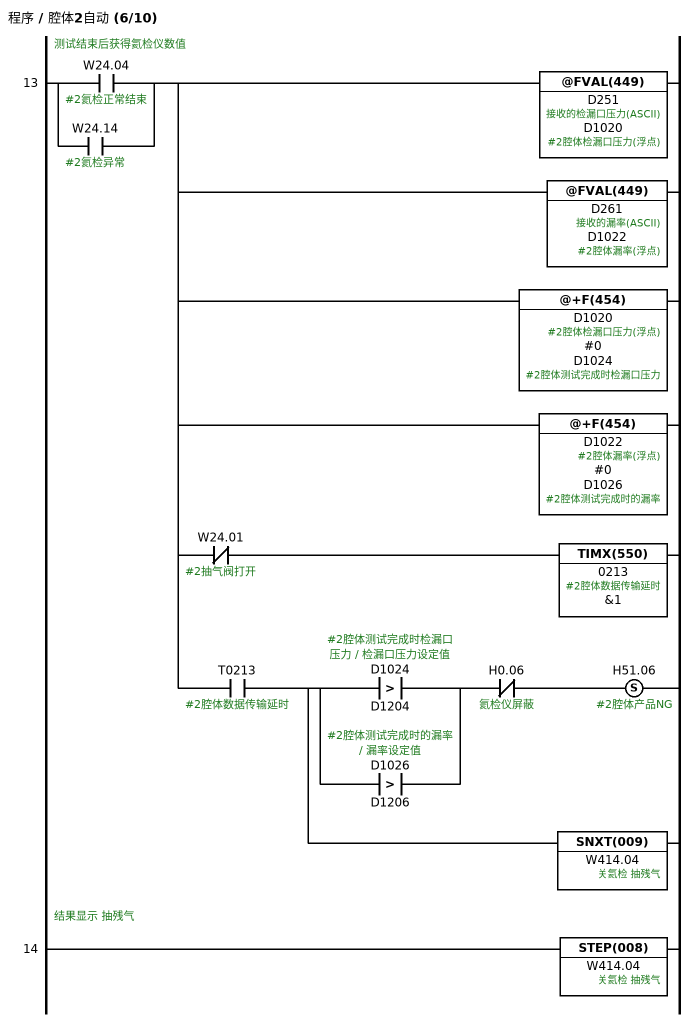
; [picture p72: 程序 / 腔体2自动, rungs 13-14]
; rung 13: 测试结束后获得氦检仪数值
LD W24.04  ; #2氦检正常结束
OR W24.14  ; #2氦检异常
OUT TR0
@FVAL(449) D251 D1020  ; 接收的检漏口压力(ASCII), #2腔体检漏口压力(浮点)
@FVAL(449) D261 D1022  ; 接收的漏率(ASCII), #2腔体漏率(浮点)
@+F(454) D1020 #0 D1024  ; #2腔体检漏口压力(浮点), #2腔体测试完成时检漏口压力
@+F(454) D1022 #0 D1026  ; #2腔体漏率(浮点), #2腔体测试完成时的漏率
ANDNOT W24.01  ; #2抽气阀打开
TIMX(550) 0213 &1  ; #2腔体数据传输延时
LD TR0
AND T0213  ; #2腔体数据传输延时
OUT TR0
LD>F(333) D1024 D1204  ; #2腔体测试完成时检漏口压力, 检漏口压力设定值
OR>F(333) D1026 D1206  ; #2腔体测试完成时的漏率, 漏率设定值
ANDLD
ANDNOT H0.06  ; 氦检仪屏蔽
SET H51.06  ; #2腔体产品NG
LD TR0
SNXT(009) W414.04  ; 关氦检 抽残气
; rung 14: 结果显示 抽残气
STEP(008) W414.04  ; 关氦检 抽残气

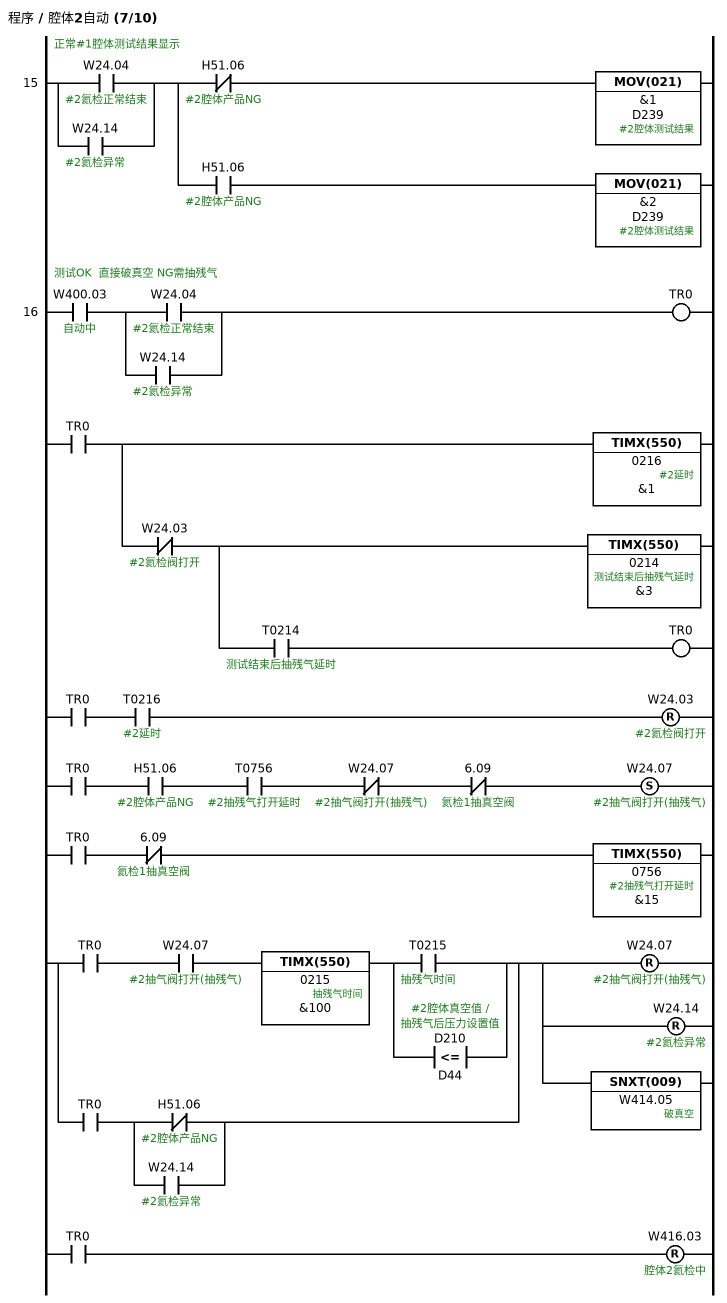
; rung 15: 正常#1腔体测试结果显示
LD W24.04  ; #2氦检正常结束
OR W24.14  ; #2氦检异常
OUT TR0
ANDNOT H51.06  ; #2腔体产品NG
MOV(021) &1 D239  ; #2腔体测试结果
LD TR0
AND H51.06  ; #2腔体产品NG
MOV(021) &2 D239  ; #2腔体测试结果
; rung 16: 测试OK  直接破真空 NG需抽残气
LD W400.03  ; 自动中
LD W24.04  ; #2氦检正常结束
OR W24.14  ; #2氦检异常
ANDLD
OUT TR0
AND T0216  ; #2延时
RSET W24.03  ; #2氦检阀打开
LD TR0
TIMX(550) 0216 &1  ; #2延时
ANDNOT W24.03  ; #2氦检阀打开
TIMX(550) 0214 &3  ; 测试结束后抽残气延时
AND T0214  ; 测试结束后抽残气延时
OUT TR0
AND H51.06  ; #2腔体产品NG
AND T0756  ; #2抽残气打开延时
ANDNOT W24.07  ; #2抽气阀打开(抽残气)
ANDNOT 6.09  ; 氦检1抽真空阀
SET W24.07  ; #2抽气阀打开(抽残气)
LD TR0
ANDNOT 6.09  ; 氦检1抽真空阀
TIMX(550) 0756 &15  ; #2抽残气打开延时
LD TR0
AND W24.07  ; #2抽气阀打开(抽残气)
TIMX(550) 0215 &100  ; 抽残气时间
LD T0215  ; 抽残气时间
OR<=F(332) D210 D44  ; #2腔体真空值, 抽残气后压力设置值
ANDLD
LD TR0
LDNOT H51.06  ; #2腔体产品NG
OR W24.14  ; #2氦检异常
ANDLD
ORLD
RSET W24.07  ; #2抽气阀打开(抽残气)
RSET W24.14  ; #2氦检异常
SNXT(009) W414.05  ; 破真空
LD TR0
RSET W416.03  ; 腔体2氦检中

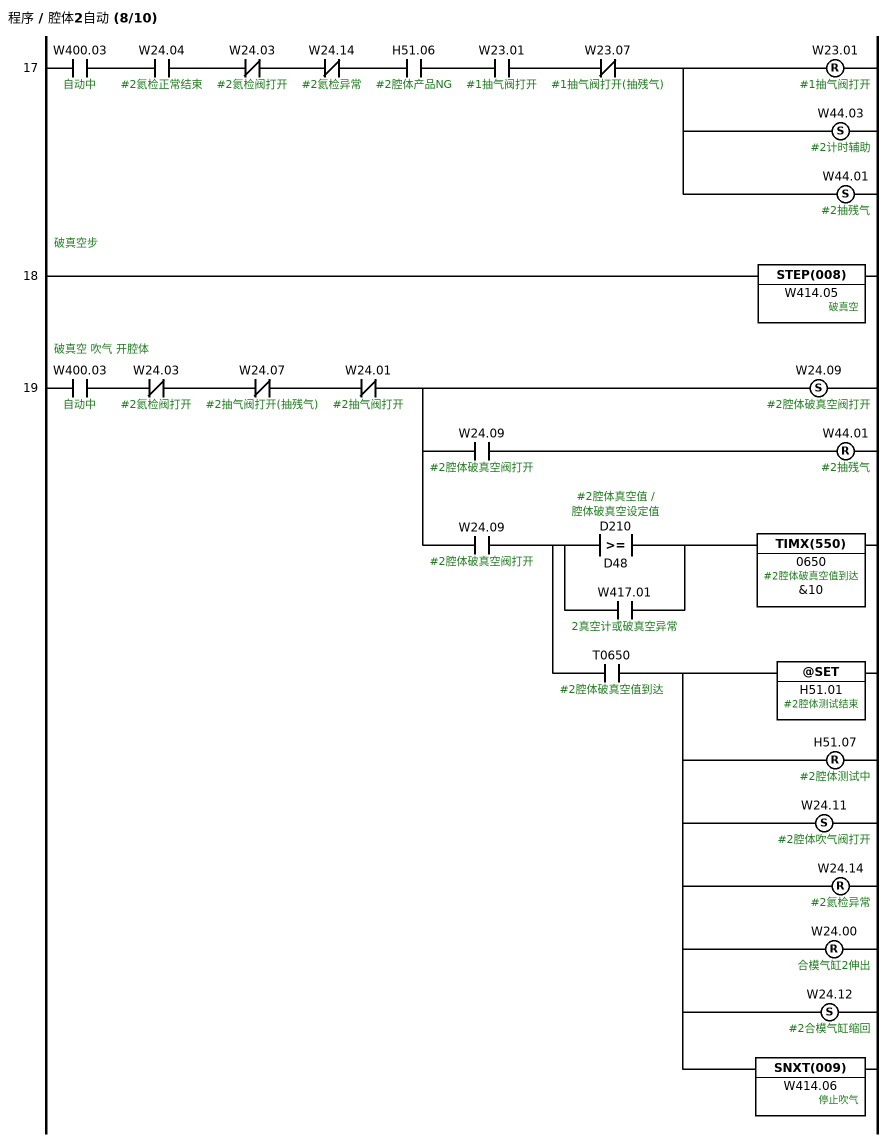
; rung 17
LD W400.03  ; 自动中
AND W24.04  ; #2氦检正常结束
ANDNOT W24.03  ; #2氦检阀打开
ANDNOT W24.14  ; #2氦检异常
AND H51.06  ; #2腔体产品NG
AND W23.01  ; #1抽气阀打开
ANDNOT W23.07  ; #1抽气阀打开(抽残气)
RSET W23.01  ; #1抽气阀打开
SET W44.03  ; #2计时辅助
SET W44.01  ; #2抽残气
; rung 18: 破真空步
STEP(008) W414.05  ; 破真空
; rung 19: 破真空 吹气 开腔体
LD W400.03  ; 自动中
ANDNOT W24.03  ; #2氦检阀打开
ANDNOT W24.07  ; #2抽气阀打开(抽残气)
ANDNOT W24.01  ; #2抽气阀打开
OUT TR0
SET W24.09  ; #2腔体破真空阀打开
AND W24.09  ; #2腔体破真空阀打开
RSET W44.01  ; #2抽残气
LD TR0
AND W24.09  ; #2腔体破真空阀打开
OUT TR0
LD>=F(334) D210 D48  ; #2腔体真空值, 腔体破真空设定值
OR W417.01  ; 2真空计或破真空异常
ANDLD
TIMX(550) 0650 &10  ; #2腔体破真空值到达
LD TR0
AND T0650  ; #2腔体破真空值到达
@SET H51.01  ; #2腔体测试结束
RSET H51.07  ; #2腔体测试中
SET W24.11  ; #2腔体吹气阀打开
RSET W24.14  ; #2氦检异常
RSET W24.00  ; 合模气缸2伸出
SET W24.12  ; #2合模气缸缩回
SNXT(009) W414.06  ; 停止吹气

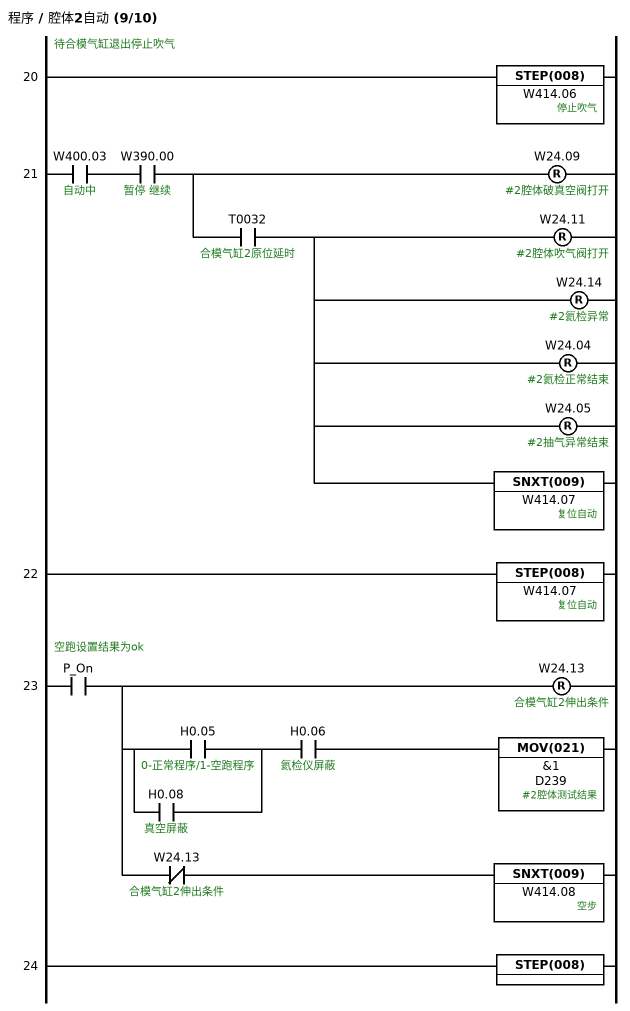
; rung 20: 待合模气缸退出停止吹气
STEP(008) W414.06  ; 停止吹气
; rung 21
LD W400.03  ; 自动中
AND W390.00  ; 暂停 继续
RSET W24.09  ; #2腔体破真空阀打开
AND T0032  ; 合模气缸2原位延时
RSET W24.11  ; #2腔体吹气阀打开
RSET W24.14  ; #2氦检异常
RSET W24.04  ; #2氦检正常结束
RSET W24.05  ; #2抽气异常结束
SNXT(009) W414.07  ; 复位自动
; rung 22
STEP(008) W414.07  ; 复位自动
; rung 23: 空跑设置结果为ok
LD P_On
OUT TR0
RSET W24.13  ; 合模气缸2伸出条件
LD H0.05  ; 0-正常程序/1-空跑程序
OR H0.08  ; 真空屏蔽
ANDLD
AND H0.06  ; 氦检仪屏蔽
MOV(021) &1 D239  ; #2腔体测试结果
LD TR0
ANDNOT W24.13  ; 合模气缸2伸出条件
SNXT(009) W414.08  ; 空步
; rung 24
STEP(008)

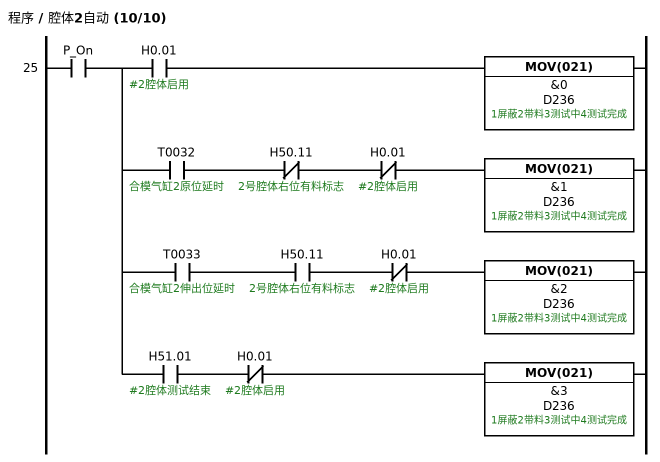
; rung 25
LD P_On
OUT TR0
AND H0.01  ; #2腔体启用
MOV(021) &0 D236  ; 1屏蔽2带料3测试中4测试完成
LD TR0
AND T0032  ; 合模气缸2原位延时
ANDNOT H50.11  ; 2号腔体右位有料标志
ANDNOT H0.01  ; #2腔体启用
MOV(021) &1 D236  ; 1屏蔽2带料3测试中4测试完成
LD TR0
AND T0033  ; 合模气缸2伸出位延时
AND H50.11  ; 2号腔体右位有料标志
ANDNOT H0.01  ; #2腔体启用
MOV(021) &2 D236  ; 1屏蔽2带料3测试中4测试完成
LD TR0
AND H51.01  ; #2腔体测试结束
ANDNOT H0.01  ; #2腔体启用
MOV(021) &3 D236  ; 1屏蔽2带料3测试中4测试完成

### Section 下料轴自动

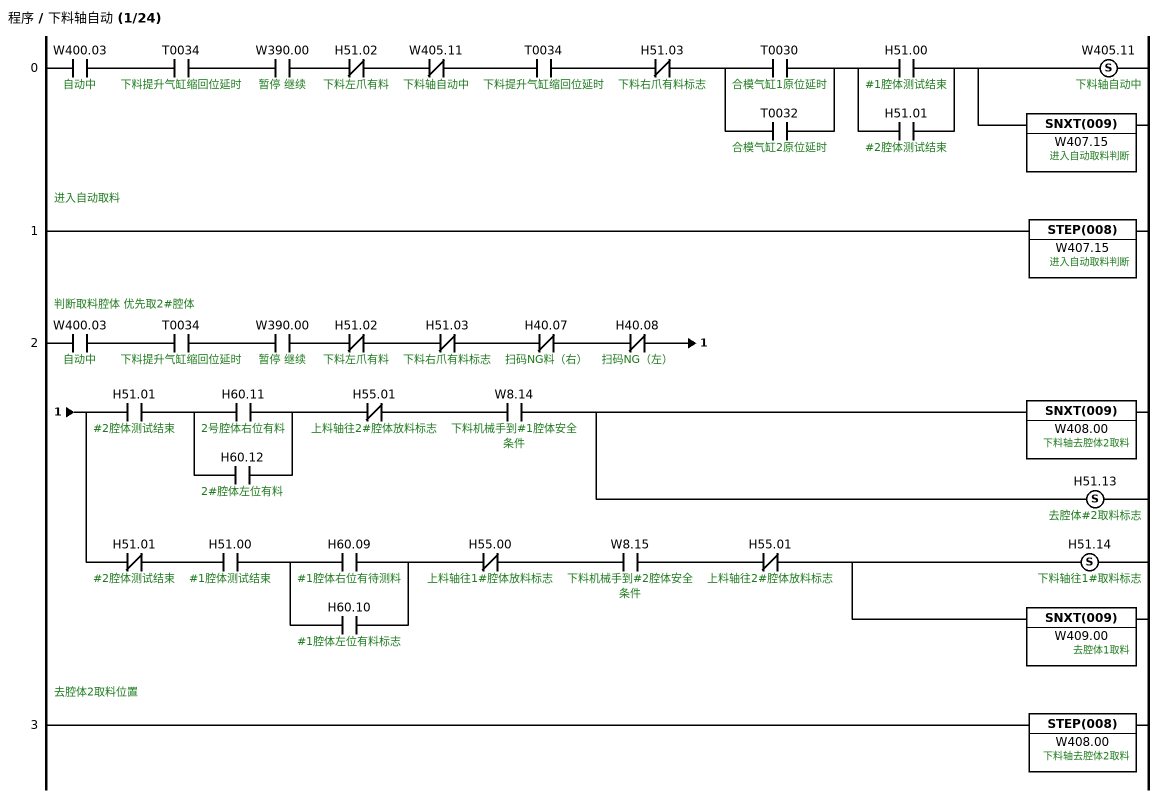
; rung 0
LD W400.03  ; 自动中
AND T0034  ; 下料提升气缸缩回位延时
AND W390.00  ; 暂停 继续
ANDNOT H51.02  ; 下料左爪有料
ANDNOT W405.11  ; 下料轴自动中
AND T0034  ; 下料提升气缸缩回位延时
ANDNOT H51.03  ; 下料右爪有料标志
LD T0030  ; 合模气缸1原位延时
OR T0032  ; 合模气缸2原位延时
ANDLD
LD H51.00  ; #1腔体测试结束
OR H51.01  ; #2腔体测试结束
ANDLD
SET W405.11  ; 下料轴自动中
SNXT(009) W407.15  ; 进入自动取料判断
; rung 1: 进入自动取料
STEP(008) W407.15  ; 进入自动取料判断
; rung 2: 判断取料腔体 优先取2#腔体
LD W400.03  ; 自动中
AND T0034  ; 下料提升气缸缩回位延时
AND W390.00  ; 暂停 继续
ANDNOT H51.02  ; 下料左爪有料
ANDNOT H51.03  ; 下料右爪有料标志
ANDNOT H40.07  ; 扫码NG料（右）
ANDNOT H40.08  ; 扫码NG（左）
OUT TR0
AND H51.01  ; #2腔体测试结束
LD H60.11  ; 2号腔体右位有料
OR H60.12  ; 2#腔体左位有料
ANDLD
ANDNOT H55.01  ; 上料轴往2#腔体放料标志
AND W8.14  ; 下料机械手到#1腔体安全条件
SNXT(009) W408.00  ; 下料轴去腔体2取料
SET H51.13  ; 去腔体#2取料标志
LD TR0
ANDNOT H51.01  ; #2腔体测试结束
AND H51.00  ; #1腔体测试结束
LD H60.09  ; #1腔体右位有待测料
OR H60.10  ; #1腔体左位有料标志
ANDLD
ANDNOT H55.00  ; 上料轴往1#腔体放料标志
AND W8.15  ; 下料机械手到#2腔体安全条件
ANDNOT H55.01  ; 上料轴往2#腔体放料标志
SET H51.14  ; 下料轴往1#取料标志
SNXT(009) W409.00  ; 去腔体1取料
; rung 3: 去腔体2取料位置
STEP(008) W408.00  ; 下料轴去腔体2取料

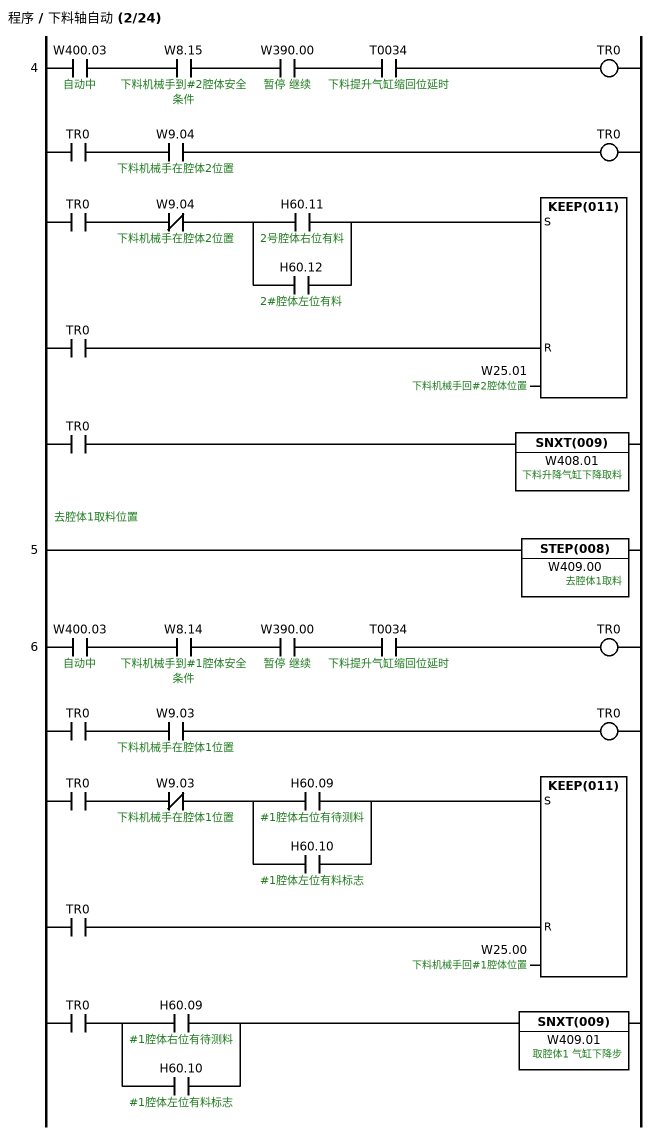
; rung 4
LD W400.03  ; 自动中
AND W8.15  ; 下料机械手到#2腔体安全条件
AND W390.00  ; 暂停 继续
AND T0034  ; 下料提升气缸缩回位延时
OUT TR0
ANDNOT W9.04  ; 下料机械手在腔体2位置
LD H60.11  ; 2号腔体右位有料
OR H60.12  ; 2#腔体左位有料
ANDLD
LD TR0
AND W9.04  ; 下料机械手在腔体2位置
OUT TR0
KEEP(011) W25.01  ; 下料机械手回#2腔体位置
LD TR0
SNXT(009) W408.01  ; 下料升降气缸下降取料
; rung 5: 去腔体1取料位置
STEP(008) W409.00  ; 去腔体1取料
; rung 6
LD W400.03  ; 自动中
AND W8.14  ; 下料机械手到#1腔体安全条件
AND W390.00  ; 暂停 继续
AND T0034  ; 下料提升气缸缩回位延时
OUT TR0
ANDNOT W9.03  ; 下料机械手在腔体1位置
LD H60.09  ; #1腔体右位有待测料
OR H60.10  ; #1腔体左位有料标志
ANDLD
LD TR0
AND W9.03  ; 下料机械手在腔体1位置
OUT TR0
KEEP(011) W25.00  ; 下料机械手回#1腔体位置
LD TR0
LD H60.09  ; #1腔体右位有待测料
OR H60.10  ; #1腔体左位有料标志
ANDLD
SNXT(009) W409.01  ; 取腔体1 气缸下降步

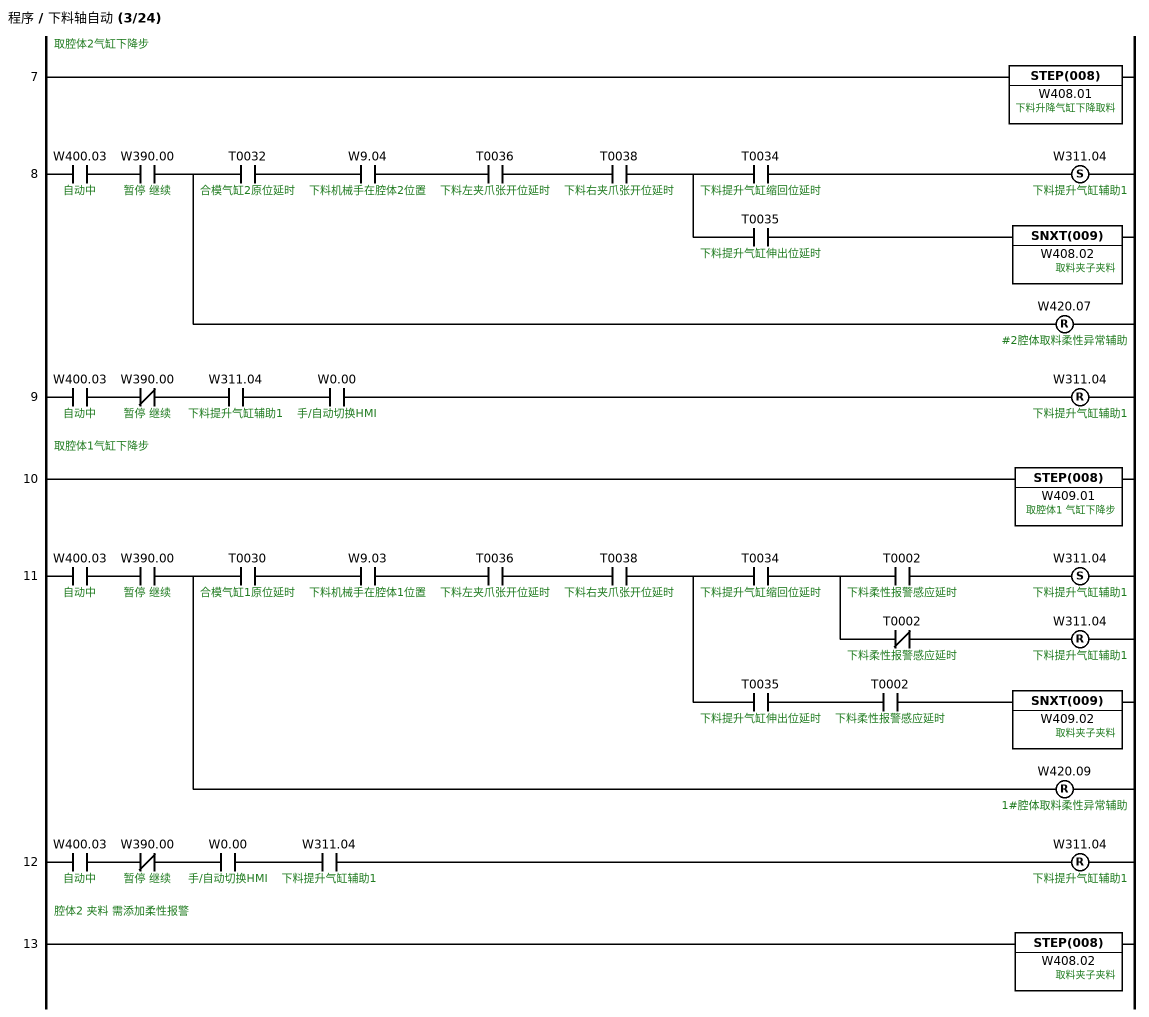
; rung 7: 取腔体2气缸下降步
STEP(008) W408.01  ; 下料升降气缸下降取料
; rung 8
LD W400.03  ; 自动中
AND W390.00  ; 暂停 继续
OUT TR0
AND T0032  ; 合模气缸2原位延时
AND W9.04  ; 下料机械手在腔体2位置
AND T0036  ; 下料左夹爪张开位延时
AND T0038  ; 下料右夹爪张开位延时
OUT TR1
AND T0034  ; 下料提升气缸缩回位延时
SET W311.04  ; 下料提升气缸辅助1
LD TR1
AND T0035  ; 下料提升气缸伸出位延时
SNXT(009) W408.02  ; 取料夹子夹料
LD TR0
RSET W420.07  ; #2腔体取料柔性异常辅助
; rung 9
LD W400.03  ; 自动中
ANDNOT W390.00  ; 暂停 继续
AND W311.04  ; 下料提升气缸辅助1
AND W0.00  ; 手/自动切换HMI
RSET W311.04  ; 下料提升气缸辅助1
; rung 10: 取腔体1气缸下降步
STEP(008) W409.01  ; 取腔体1 气缸下降步
; rung 11
LD W400.03  ; 自动中
AND W390.00  ; 暂停 继续
OUT TR0
AND T0030  ; 合模气缸1原位延时
AND W9.03  ; 下料机械手在腔体1位置
AND T0036  ; 下料左夹爪张开位延时
AND T0038  ; 下料右夹爪张开位延时
OUT TR1
AND T0034  ; 下料提升气缸缩回位延时
OUT TR2
AND T0002  ; 下料柔性报警感应延时
SET W311.04  ; 下料提升气缸辅助1
LD TR2
ANDNOT T0002  ; 下料柔性报警感应延时
RSET W311.04  ; 下料提升气缸辅助1
LD TR1
AND T0035  ; 下料提升气缸伸出位延时
AND T0002  ; 下料柔性报警感应延时
SNXT(009) W409.02  ; 取料夹子夹料
LD TR0
RSET W420.09  ; 1#腔体取料柔性异常辅助
; rung 12
LD W400.03  ; 自动中
ANDNOT W390.00  ; 暂停 继续
AND W0.00  ; 手/自动切换HMI
AND W311.04  ; 下料提升气缸辅助1
RSET W311.04  ; 下料提升气缸辅助1
; rung 13: 腔体2 夹料 需添加柔性报警
STEP(008) W408.02  ; 取料夹子夹料

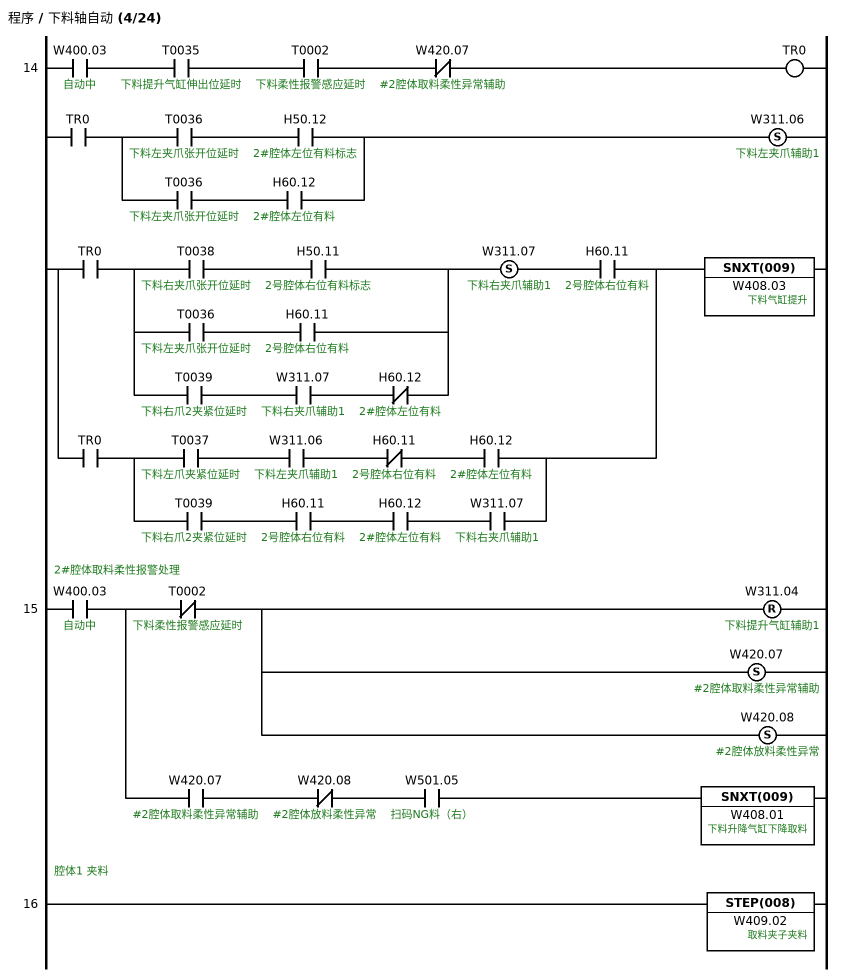
; rung 14
LD W400.03  ; 自动中
AND T0035  ; 下料提升气缸伸出位延时
AND T0002  ; 下料柔性报警感应延时
ANDNOT W420.07  ; #2腔体取料柔性异常辅助
OUT TR0
LD T0036  ; 下料左夹爪张开位延时
AND H50.12  ; 2#腔体左位有料标志
LD T0036  ; 下料左夹爪张开位延时
AND H60.12  ; 2#腔体左位有料
ORLD
ANDLD
SET W311.06  ; 下料左夹爪辅助1
LD TR0
LD T0038  ; 下料右夹爪张开位延时
AND H50.11  ; 2号腔体右位有料标志
LD T0036  ; 下料左夹爪张开位延时
AND H60.11  ; 2号腔体右位有料
ORLD
LD T0039  ; 下料右爪2夹紧位延时
AND W311.07  ; 下料右夹爪辅助1
ANDNOT H60.12  ; 2#腔体左位有料
ORLD
ANDLD
SET W311.07  ; 下料右夹爪辅助1
AND H60.11  ; 2号腔体右位有料
LD TR0
LD T0037  ; 下料左爪夹紧位延时
AND W311.06  ; 下料左夹爪辅助1
ANDNOT H60.11  ; 2号腔体右位有料
AND H60.12  ; 2#腔体左位有料
LD T0039  ; 下料右爪2夹紧位延时
AND H60.11  ; 2号腔体右位有料
AND H60.12  ; 2#腔体左位有料
AND W311.07  ; 下料右夹爪辅助1
ORLD
ANDLD
ORLD
SNXT(009) W408.03  ; 下料气缸提升
; rung 15: 2#腔体取料柔性报警处理
LD W400.03  ; 自动中
OUT TR0
ANDNOT T0002  ; 下料柔性报警感应延时
RSET W311.04  ; 下料提升气缸辅助1
SET W420.07  ; #2腔体取料柔性异常辅助
SET W420.08  ; #2腔体放料柔性异常
LD TR0
AND W420.07  ; #2腔体取料柔性异常辅助
ANDNOT W420.08  ; #2腔体放料柔性异常
AND W501.05  ; 扫码NG料（右）
SNXT(009) W408.01  ; 下料升降气缸下降取料
; rung 16: 腔体1 夹料
STEP(008) W409.02  ; 取料夹子夹料

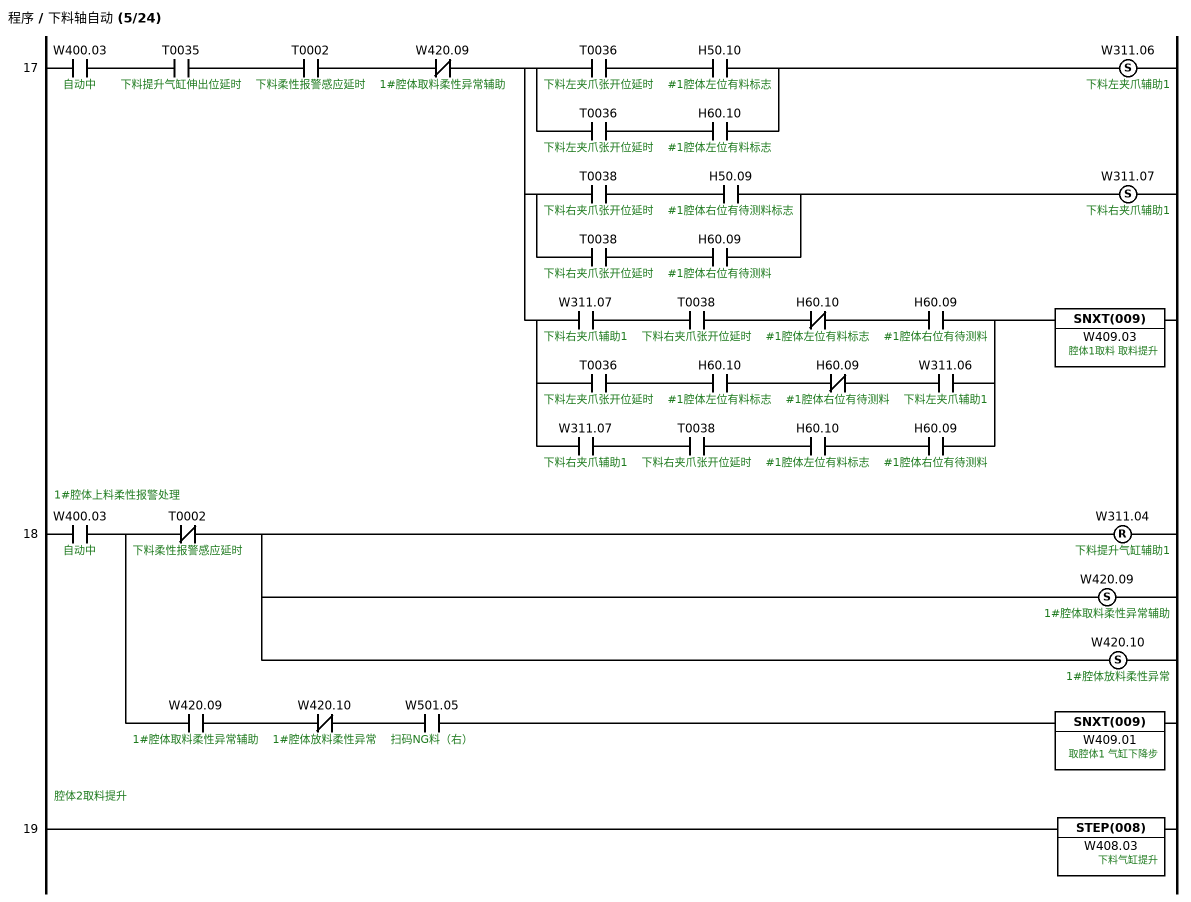
; rung 17
LD W400.03  ; 自动中
AND T0035  ; 下料提升气缸伸出位延时
AND T0002  ; 下料柔性报警感应延时
ANDNOT W420.09  ; 1#腔体取料柔性异常辅助
OUT TR0
LD T0036  ; 下料左夹爪张开位延时
AND H50.10  ; #1腔体左位有料标志
LD T0036  ; 下料左夹爪张开位延时
AND H60.10  ; #1腔体左位有料标志
ORLD
ANDLD
SET W311.06  ; 下料左夹爪辅助1
LD TR0
LD T0038  ; 下料右夹爪张开位延时
AND H50.09  ; #1腔体右位有待测料标志
LD T0038  ; 下料右夹爪张开位延时
AND H60.09  ; #1腔体右位有待测料
ORLD
ANDLD
SET W311.07  ; 下料右夹爪辅助1
LD TR0
LD W311.07  ; 下料右夹爪辅助1
AND T0038  ; 下料右夹爪张开位延时
ANDNOT H60.10  ; #1腔体左位有料标志
AND H60.09  ; #1腔体右位有待测料
LD T0036  ; 下料左夹爪张开位延时
AND H60.10  ; #1腔体左位有料标志
ANDNOT H60.09  ; #1腔体右位有待测料
AND W311.06  ; 下料左夹爪辅助1
ORLD
LD W311.07  ; 下料右夹爪辅助1
AND T0038  ; 下料右夹爪张开位延时
AND H60.10  ; #1腔体左位有料标志
AND H60.09  ; #1腔体右位有待测料
ORLD
ANDLD
SNXT(009) W409.03  ; 腔体1取料 取料提升
; rung 18: 1#腔体上料柔性报警处理
LD W400.03  ; 自动中
OUT TR0
ANDNOT T0002  ; 下料柔性报警感应延时
RSET W311.04  ; 下料提升气缸辅助1
SET W420.09  ; 1#腔体取料柔性异常辅助
SET W420.10  ; 1#腔体放料柔性异常
LD TR0
AND W420.09  ; 1#腔体取料柔性异常辅助
ANDNOT W420.10  ; 1#腔体放料柔性异常
AND W501.05  ; 扫码NG料（右）
SNXT(009) W409.01  ; 取腔体1 气缸下降步
; rung 19: 腔体2取料提升
STEP(008) W408.03  ; 下料气缸提升

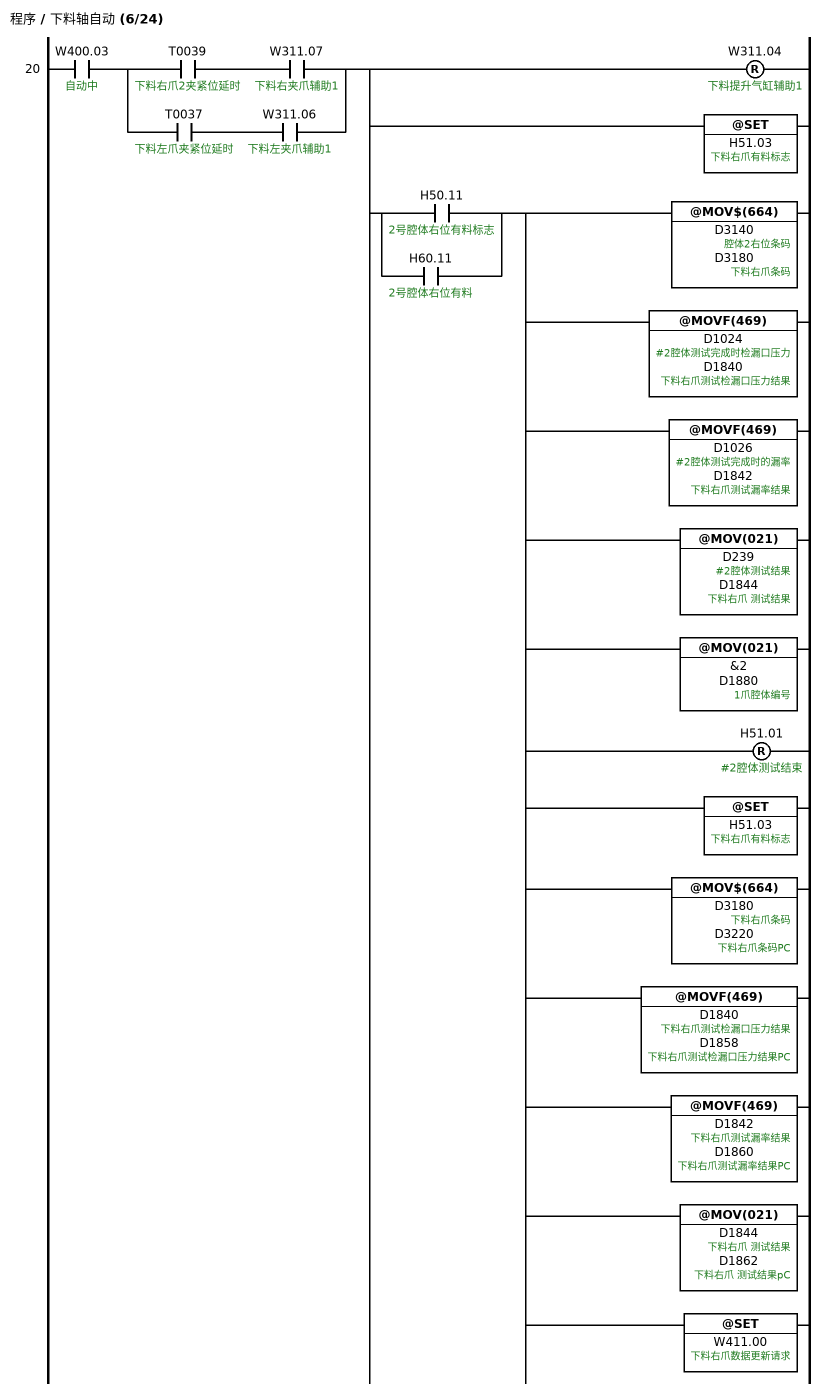

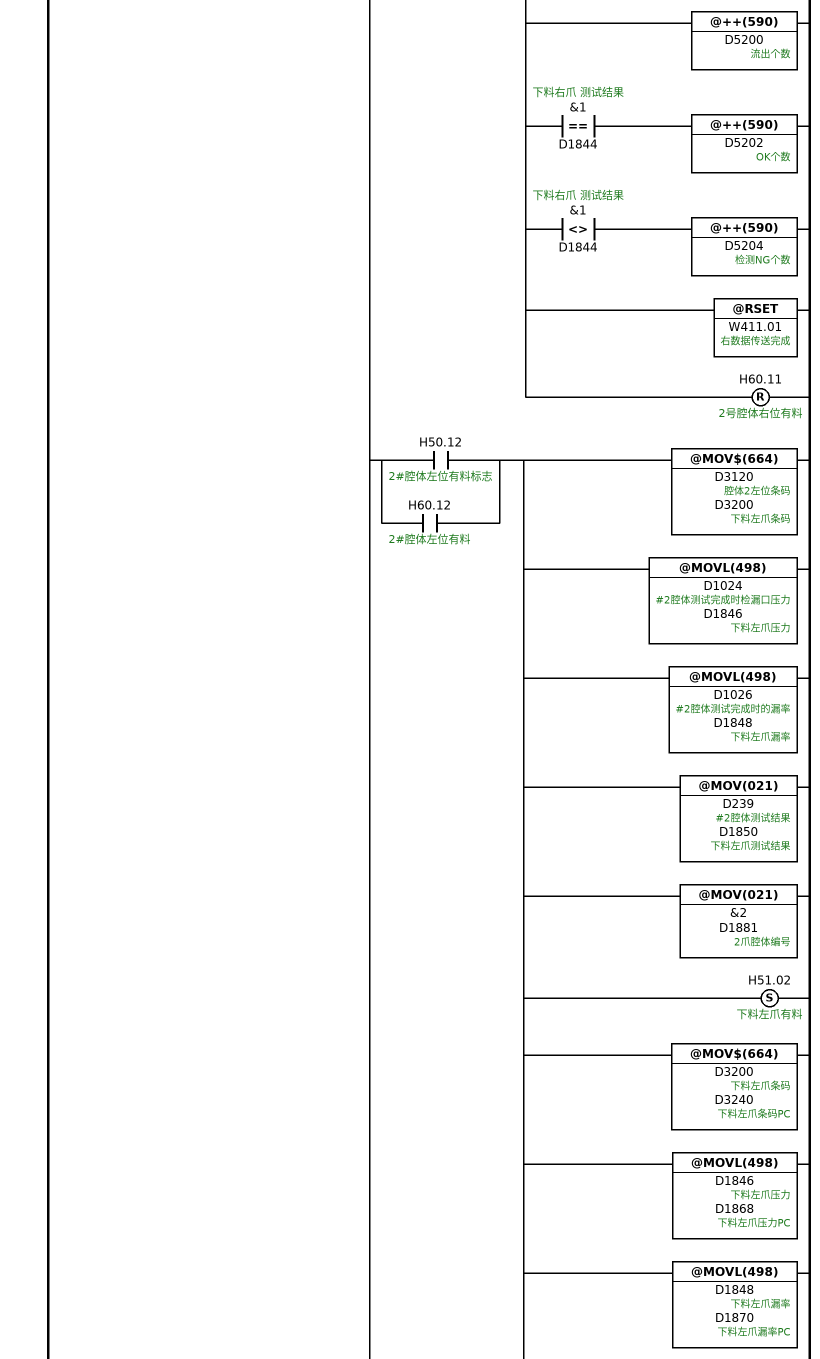

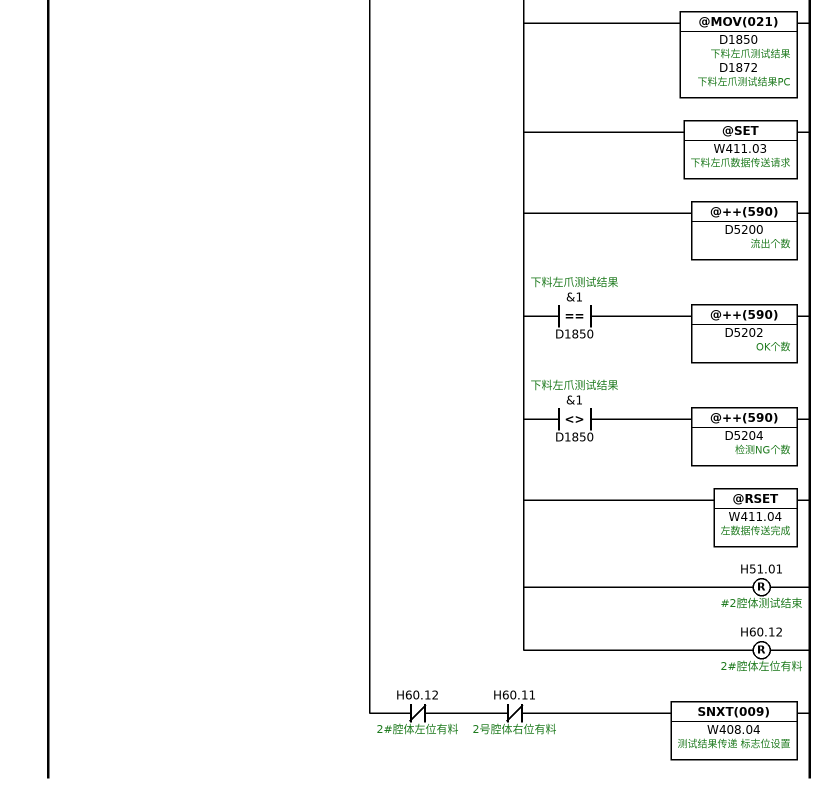
; rung 20
LD W400.03  ; 自动中
LD T0039  ; 下料右爪2夹紧位延时
AND W311.07  ; 下料右夹爪辅助1
LD T0037  ; 下料左爪夹紧位延时
AND W311.06  ; 下料左夹爪辅助1
ORLD
ANDLD
OUT TR0
RSET W311.04  ; 下料提升气缸辅助1
@SET H51.03  ; 下料右爪有料标志
LD H50.11  ; 2号腔体右位有料标志
OR H60.11  ; 2号腔体右位有料
ANDLD
OUT TR1
@MOV$(664) D3140 D3180  ; 腔体2右位条码, 下料右爪条码
@MOVF(469) D1024 D1840  ; #2腔体测试完成时检漏口压力, 下料右爪测试检漏口压力结果
@MOVF(469) D1026 D1842  ; #2腔体测试完成时的漏率, 下料右爪测试漏率结果
@MOV(021) D239 D1844  ; #2腔体测试结果, 下料右爪 测试结果
@MOV(021) &2 D1880  ; 1爪腔体编号
RSET H51.01  ; #2腔体测试结束
@SET H51.03  ; 下料右爪有料标志
@MOV$(664) D3180 D3220  ; 下料右爪条码, 下料右爪条码PC
@MOVF(469) D1840 D1858  ; 下料右爪测试检漏口压力结果, 下料右爪测试检漏口压力结果PC
@MOVF(469) D1842 D1860  ; 下料右爪测试漏率结果, 下料右爪测试漏率结果PC
@MOV(021) D1844 D1862  ; 下料右爪 测试结果, 下料右爪 测试结果pC
@SET W411.00  ; 下料右爪数据更新请求
@++(590) D5200  ; 流出个数
AND=(300) &1 D1844  ; 下料右爪 测试结果
@++(590) D5202  ; OK个数
LD TR1
AND<>(305) &1 D1844  ; 下料右爪 测试结果
@++(590) D5204  ; 检测NG个数
LD TR1
@RSET W411.01  ; 右数据传送完成
RSET H60.11  ; 2号腔体右位有料
LD TR0
LD H50.12  ; 2#腔体左位有料标志
OR H60.12  ; 2#腔体左位有料
ANDLD
OUT TR1
@MOV$(664) D3120 D3200  ; 腔体2左位条码, 下料左爪条码
@MOVL(498) D1024 D1846  ; #2腔体测试完成时检漏口压力, 下料左爪压力
@MOVL(498) D1026 D1848  ; #2腔体测试完成时的漏率, 下料左爪漏率
@MOV(021) D239 D1850  ; #2腔体测试结果, 下料左爪测试结果
@MOV(021) &2 D1881  ; 2爪腔体编号
SET H51.02  ; 下料左爪有料
@MOV$(664) D3200 D3240  ; 下料左爪条码, 下料左爪条码PC
@MOVL(498) D1846 D1868  ; 下料左爪压力, 下料左爪压力PC
@MOVL(498) D1848 D1870  ; 下料左爪漏率, 下料左爪漏率PC
@MOV(021) D1850 D1872  ; 下料左爪测试结果, 下料左爪测试结果PC
@SET W411.03  ; 下料左爪数据传送请求
@++(590) D5200  ; 流出个数
AND=(300) &1 D1850  ; 下料左爪测试结果
@++(590) D5202  ; OK个数
LD TR1
AND<>(305) &1 D1850  ; 下料左爪测试结果
@++(590) D5204  ; 检测NG个数
LD TR1
@RSET W411.04  ; 左数据传送完成
RSET H51.01  ; #2腔体测试结束
RSET H60.12  ; 2#腔体左位有料
LD TR0
ANDNOT H60.12  ; 2#腔体左位有料
ANDNOT H60.11  ; 2号腔体右位有料
SNXT(009) W408.04  ; 测试结果传递 标志位设置

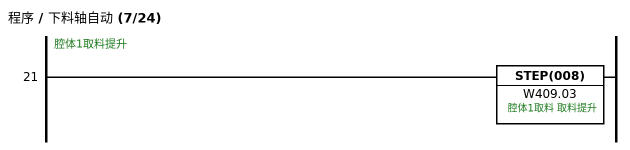
; rung 21: 腔体1取料提升
STEP(008) W409.03  ; 腔体1取料 取料提升

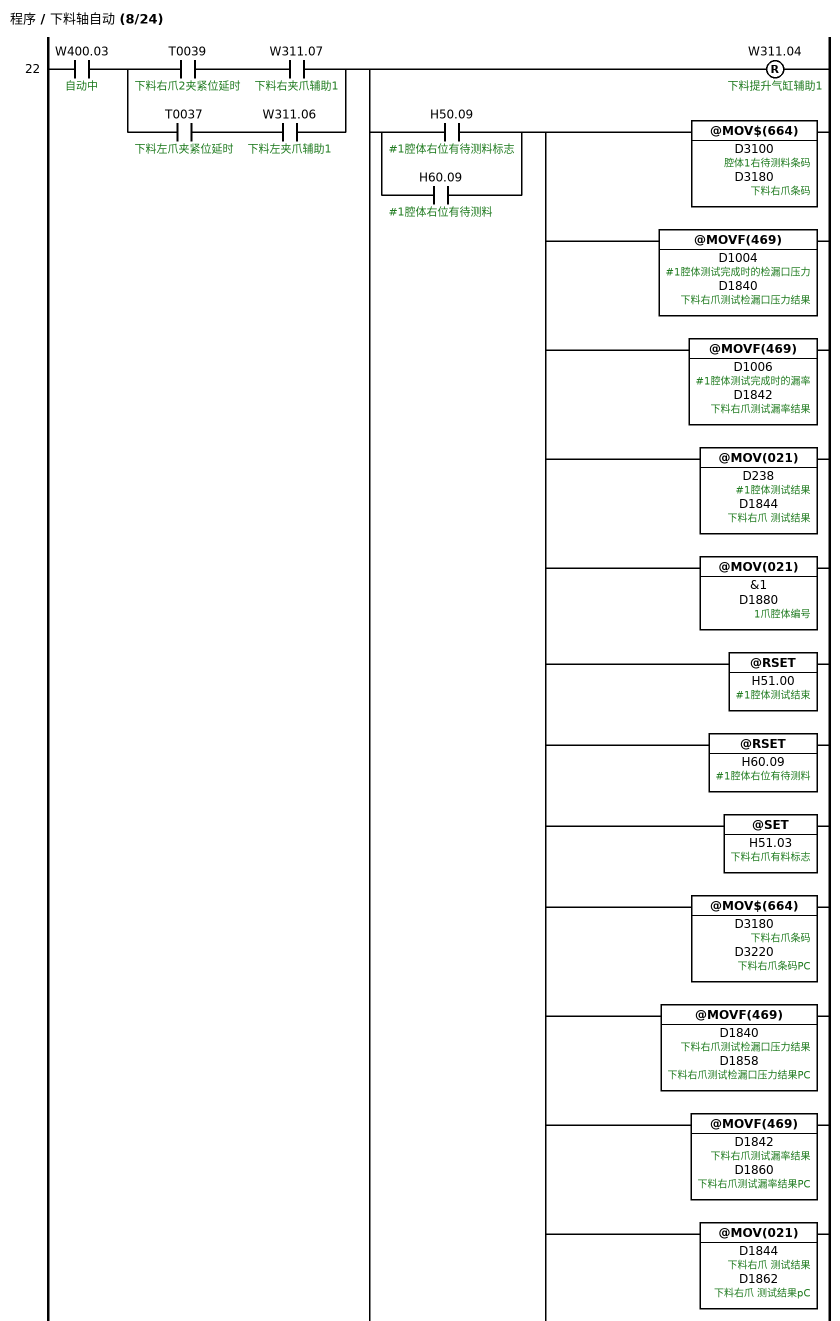

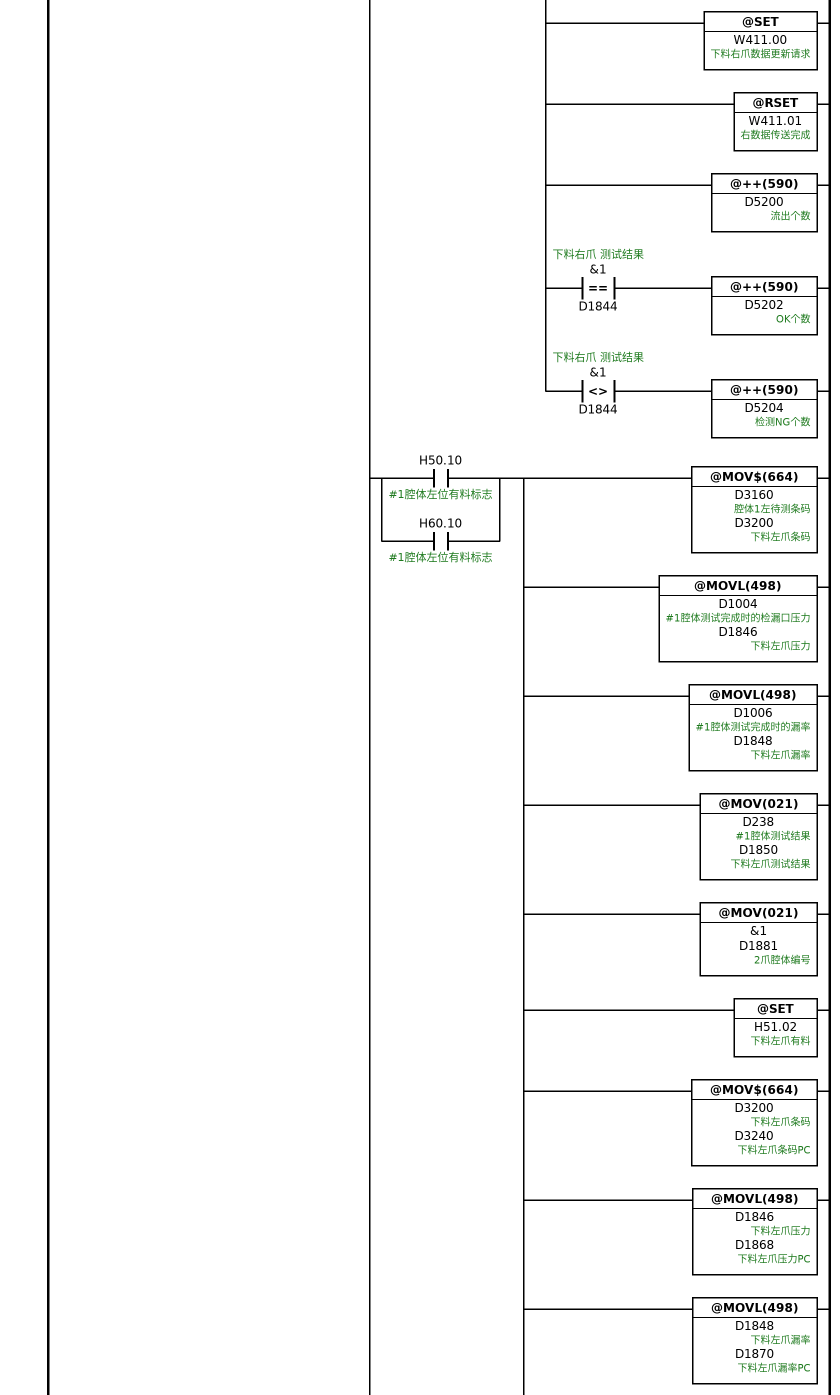

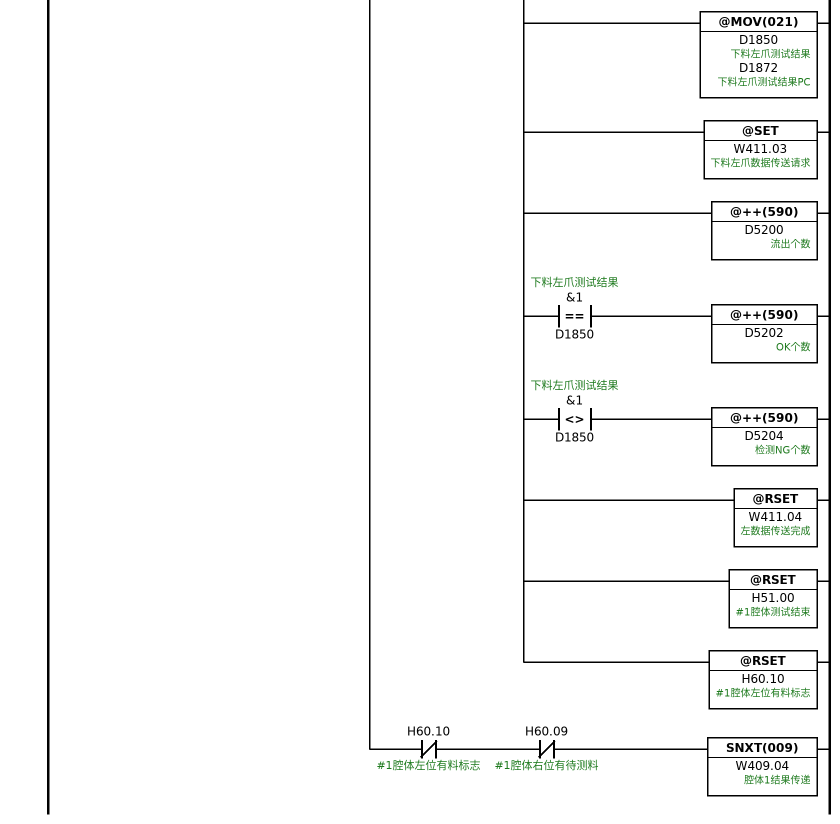
; rung 22
LD W400.03  ; 自动中
LD T0039  ; 下料右爪2夹紧位延时
AND W311.07  ; 下料右夹爪辅助1
LD T0037  ; 下料左爪夹紧位延时
AND W311.06  ; 下料左夹爪辅助1
ORLD
ANDLD
OUT TR0
RSET W311.04  ; 下料提升气缸辅助1
LD H50.09  ; #1腔体右位有待测料标志
OR H60.09  ; #1腔体右位有待测料
ANDLD
OUT TR1
@MOV$(664) D3100 D3180  ; 腔体1右待测料条码, 下料右爪条码
@MOVF(469) D1004 D1840  ; #1腔体测试完成时的检漏口压力, 下料右爪测试检漏口压力结果
@MOVF(469) D1006 D1842  ; #1腔体测试完成时的漏率, 下料右爪测试漏率结果
@MOV(021) D238 D1844  ; #1腔体测试结果, 下料右爪 测试结果
@MOV(021) &1 D1880  ; 1爪腔体编号
@RSET H51.00  ; #1腔体测试结束
@RSET H60.09  ; #1腔体右位有待测料
@SET H51.03  ; 下料右爪有料标志
@MOV$(664) D3180 D3220  ; 下料右爪条码, 下料右爪条码PC
@MOVF(469) D1840 D1858  ; 下料右爪测试检漏口压力结果, 下料右爪测试检漏口压力结果PC
@MOVF(469) D1842 D1860  ; 下料右爪测试漏率结果, 下料右爪测试漏率结果PC
@MOV(021) D1844 D1862  ; 下料右爪 测试结果, 下料右爪 测试结果pC
@SET W411.00  ; 下料右爪数据更新请求
@RSET W411.01  ; 右数据传送完成
@++(590) D5200  ; 流出个数
AND=(300) &1 D1844  ; 下料右爪 测试结果
@++(590) D5202  ; OK个数
LD TR1
AND<>(305) &1 D1844  ; 下料右爪 测试结果
@++(590) D5204  ; 检测NG个数
LD TR0
LD H50.10  ; #1腔体左位有料标志
OR H60.10  ; #1腔体左位有料标志
ANDLD
OUT TR1
@MOV$(664) D3160 D3200  ; 腔体1左待测条码, 下料左爪条码
@MOVL(498) D1004 D1846  ; #1腔体测试完成时的检漏口压力, 下料左爪压力
@MOVL(498) D1006 D1848  ; #1腔体测试完成时的漏率, 下料左爪漏率
@MOV(021) D238 D1850  ; #1腔体测试结果, 下料左爪测试结果
@MOV(021) &1 D1881  ; 2爪腔体编号
@SET H51.02  ; 下料左爪有料
@MOV$(664) D3200 D3240  ; 下料左爪条码, 下料左爪条码PC
@MOVL(498) D1846 D1868  ; 下料左爪压力, 下料左爪压力PC
@MOVL(498) D1848 D1870  ; 下料左爪漏率, 下料左爪漏率PC
@MOV(021) D1850 D1872  ; 下料左爪测试结果, 下料左爪测试结果PC
@SET W411.03  ; 下料左爪数据传送请求
@++(590) D5200  ; 流出个数
AND=(300) &1 D1850  ; 下料左爪测试结果
@++(590) D5202  ; OK个数
LD TR1
AND<>(305) &1 D1850  ; 下料左爪测试结果
@++(590) D5204  ; 检测NG个数
LD TR1
@RSET W411.04  ; 左数据传送完成
@RSET H51.00  ; #1腔体测试结束
@RSET H60.10  ; #1腔体左位有料标志
LD TR0
ANDNOT H60.10  ; #1腔体左位有料标志
ANDNOT H60.09  ; #1腔体右位有待测料
SNXT(009) W409.04  ; 腔体1结果传递

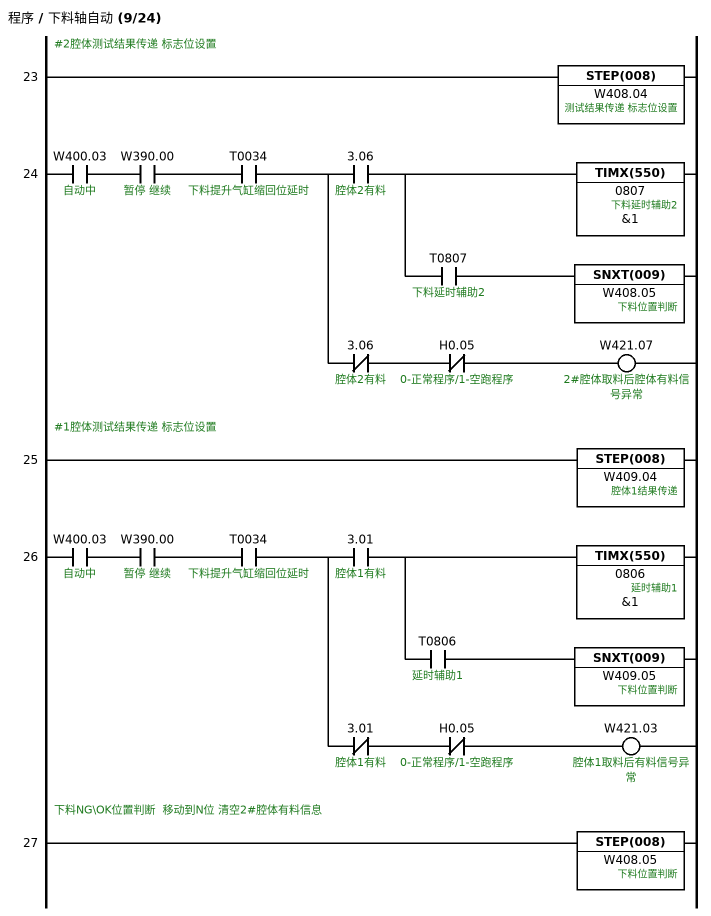
; rung 23: #2腔体测试结果传递 标志位设置
STEP(008) W408.04  ; 测试结果传递 标志位设置
; rung 24
LD W400.03  ; 自动中
AND W390.00  ; 暂停 继续
AND T0034  ; 下料提升气缸缩回位延时
OUT TR0
AND 3.06  ; 腔体2有料
TIMX(550) 0807 &1  ; 下料延时辅助2
AND T0807  ; 下料延时辅助2
SNXT(009) W408.05  ; 下料位置判断
LD TR0
ANDNOT 3.06  ; 腔体2有料
ANDNOT H0.05  ; 0-正常程序/1-空跑程序
OUT W421.07  ; 2#腔体取料后腔体有料信号异常
; rung 25: #1腔体测试结果传递 标志位设置
STEP(008) W409.04  ; 腔体1结果传递
; rung 26
LD W400.03  ; 自动中
AND W390.00  ; 暂停 继续
AND T0034  ; 下料提升气缸缩回位延时
OUT TR0
AND 3.01  ; 腔体1有料
TIMX(550) 0806 &1  ; 延时辅助1
AND T0806  ; 延时辅助1
SNXT(009) W409.05  ; 下料位置判断
LD TR0
ANDNOT 3.01  ; 腔体1有料
ANDNOT H0.05  ; 0-正常程序/1-空跑程序
OUT W421.03  ; 腔体1取料后有料信号异常
; rung 27: 下料NG\OK位置判断  移动到N位 清空2#腔体有料信息
STEP(008) W408.05  ; 下料位置判断

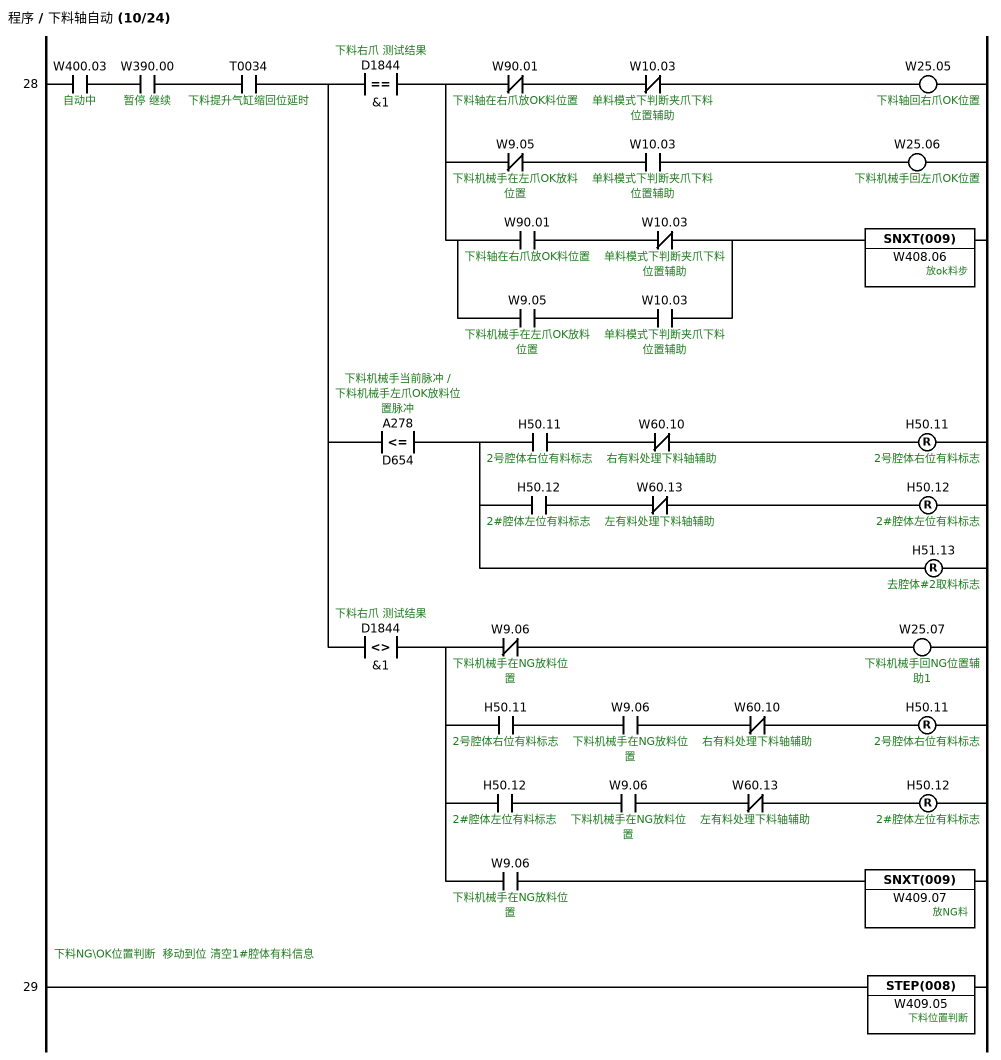
; rung 28
LD W400.03  ; 自动中
AND W390.00  ; 暂停 继续
AND T0034  ; 下料提升气缸缩回位延时
OUT TR0
AND=(300) D1844 &1  ; 下料右爪 测试结果
OUT TR1
ANDNOT W90.01  ; 下料轴在右爪放OK料位置
ANDNOT W10.03  ; 单料模式下判断夹爪下料位置辅助
OUT W25.05  ; 下料轴回右爪OK位置
LD TR1
ANDNOT W9.05  ; 下料机械手在左爪OK放料位置
AND W10.03  ; 单料模式下判断夹爪下料位置辅助
OUT W25.06  ; 下料机械手回左爪OK位置
LD TR1
LD W90.01  ; 下料轴在右爪放OK料位置
ANDNOT W10.03  ; 单料模式下判断夹爪下料位置辅助
LD W9.05  ; 下料机械手在左爪OK放料位置
AND W10.03  ; 单料模式下判断夹爪下料位置辅助
ORLD
ANDLD
SNXT(009) W408.06  ; 放ok料步
LD TR0
AND<=SL(318) A278 D654  ; 下料机械手当前脉冲, 下料机械手左爪OK放料位置脉冲
OUT TR1
AND H50.11  ; 2号腔体右位有料标志
ANDNOT W60.10  ; 右有料处理下料轴辅助
RSET H50.11  ; 2号腔体右位有料标志
LD TR1
AND H50.12  ; 2#腔体左位有料标志
ANDNOT W60.13  ; 左有料处理下料轴辅助
RSET H50.12  ; 2#腔体左位有料标志
LD TR1
RSET H51.13  ; 去腔体#2取料标志
LD TR0
AND<>(305) D1844 &1  ; 下料右爪 测试结果
OUT TR0
ANDNOT W9.06  ; 下料机械手在NG放料位置
OUT W25.07  ; 下料机械手回NG位置辅助1
LD TR0
AND H50.11  ; 2号腔体右位有料标志
AND W9.06  ; 下料机械手在NG放料位置
ANDNOT W60.10  ; 右有料处理下料轴辅助
RSET H50.11  ; 2号腔体右位有料标志
LD TR0
AND H50.12  ; 2#腔体左位有料标志
AND W9.06  ; 下料机械手在NG放料位置
ANDNOT W60.13  ; 左有料处理下料轴辅助
RSET H50.12  ; 2#腔体左位有料标志
LD TR0
AND W9.06  ; 下料机械手在NG放料位置
SNXT(009) W409.07  ; 放NG料
; rung 29: 下料NG\OK位置判断  移动到位 清空1#腔体有料信息
STEP(008) W409.05  ; 下料位置判断

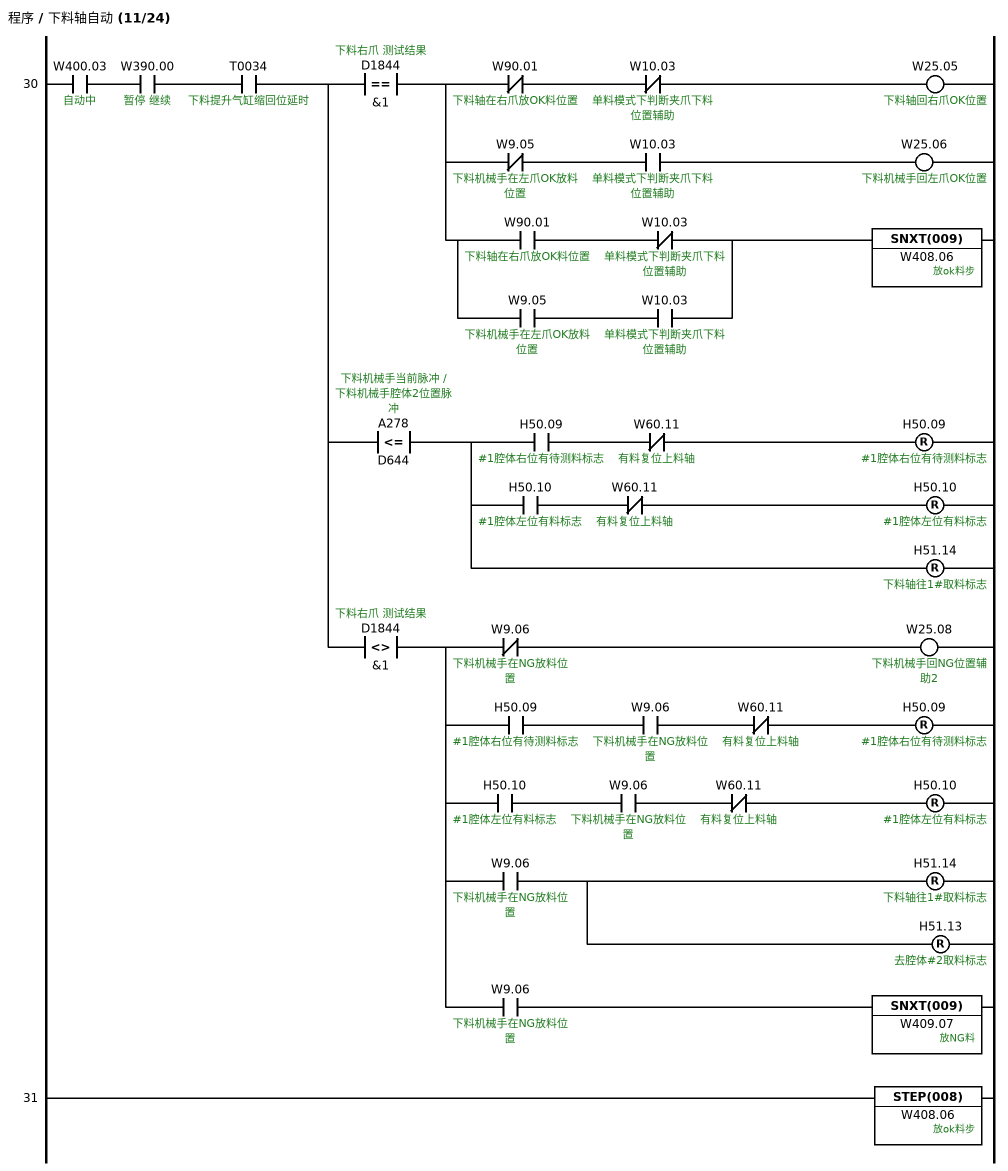
; rung 30
LD W400.03  ; 自动中
AND W390.00  ; 暂停 继续
AND T0034  ; 下料提升气缸缩回位延时
OUT TR0
AND=(300) D1844 &1  ; 下料右爪 测试结果
OUT TR1
ANDNOT W90.01  ; 下料轴在右爪放OK料位置
ANDNOT W10.03  ; 单料模式下判断夹爪下料位置辅助
OUT W25.05  ; 下料轴回右爪OK位置
LD TR1
ANDNOT W9.05  ; 下料机械手在左爪OK放料位置
AND W10.03  ; 单料模式下判断夹爪下料位置辅助
OUT W25.06  ; 下料机械手回左爪OK位置
LD TR1
LD W90.01  ; 下料轴在右爪放OK料位置
ANDNOT W10.03  ; 单料模式下判断夹爪下料位置辅助
LD W9.05  ; 下料机械手在左爪OK放料位置
AND W10.03  ; 单料模式下判断夹爪下料位置辅助
ORLD
ANDLD
SNXT(009) W408.06  ; 放ok料步
LD TR0
AND<=SL(318) A278 D644  ; 下料机械手当前脉冲, 下料机械手腔体2位置脉冲
OUT TR1
AND H50.09  ; #1腔体右位有待测料标志
ANDNOT W60.11  ; 有料复位上料轴
RSET H50.09  ; #1腔体右位有待测料标志
LD TR1
AND H50.10  ; #1腔体左位有料标志
ANDNOT W60.11  ; 有料复位上料轴
RSET H50.10  ; #1腔体左位有料标志
LD TR1
RSET H51.14  ; 下料轴往1#取料标志
LD TR0
AND<>(305) D1844 &1  ; 下料右爪 测试结果
OUT TR0
ANDNOT W9.06  ; 下料机械手在NG放料位置
OUT W25.08  ; 下料机械手回NG位置辅助2
LD TR0
AND H50.09  ; #1腔体右位有待测料标志
AND W9.06  ; 下料机械手在NG放料位置
ANDNOT W60.11  ; 有料复位上料轴
RSET H50.09  ; #1腔体右位有待测料标志
LD TR0
AND H50.10  ; #1腔体左位有料标志
AND W9.06  ; 下料机械手在NG放料位置
ANDNOT W60.11  ; 有料复位上料轴
RSET H50.10  ; #1腔体左位有料标志
LD TR0
AND W9.06  ; 下料机械手在NG放料位置
RSET H51.14  ; 下料轴往1#取料标志
RSET H51.13  ; 去腔体#2取料标志
LD TR0
AND W9.06  ; 下料机械手在NG放料位置
SNXT(009) W409.07  ; 放NG料
; rung 31
STEP(008) W408.06  ; 放ok料步

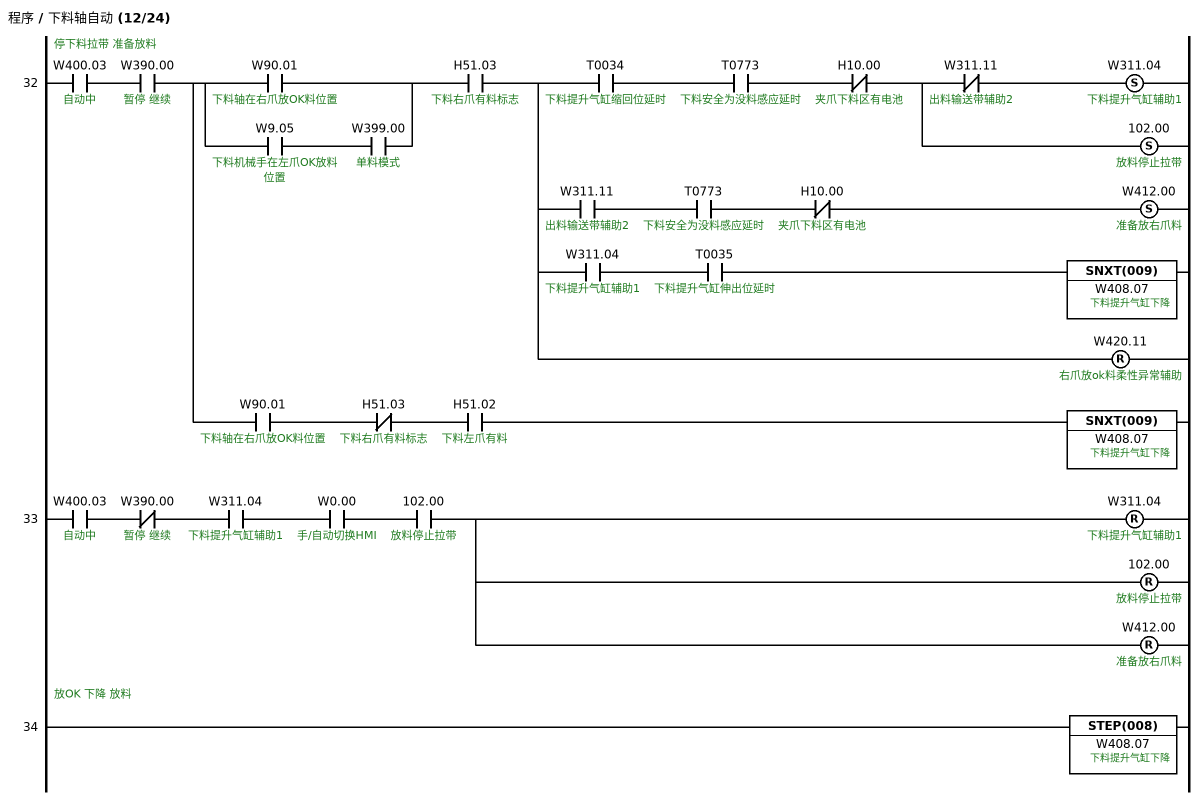
; rung 32: 停下料拉带 准备放料
LD W400.03  ; 自动中
AND W390.00  ; 暂停 继续
OUT TR0
LD W90.01  ; 下料轴在右爪放OK料位置
LD W9.05  ; 下料机械手在左爪OK放料位置
AND W399.00  ; 单料模式
ORLD
ANDLD
AND H51.03  ; 下料右爪有料标志
OUT TR1
AND T0034  ; 下料提升气缸缩回位延时
AND T0773  ; 下料安全为没料感应延时
ANDNOT H10.00  ; 夹爪下料区有电池
OUT TR2
ANDNOT W311.11  ; 出料输送带辅助2
SET W311.04  ; 下料提升气缸辅助1
LD TR2
SET 102.00  ; 放料停止拉带
LD TR1
AND W311.11  ; 出料输送带辅助2
AND T0773  ; 下料安全为没料感应延时
ANDNOT H10.00  ; 夹爪下料区有电池
SET W412.00  ; 准备放右爪料
LD TR1
AND W311.04  ; 下料提升气缸辅助1
AND T0035  ; 下料提升气缸伸出位延时
SNXT(009) W408.07  ; 下料提升气缸下降
LD TR1
RSET W420.11  ; 右爪放ok料柔性异常辅助
LD TR0
AND W90.01  ; 下料轴在右爪放OK料位置
ANDNOT H51.03  ; 下料右爪有料标志
AND H51.02  ; 下料左爪有料
SNXT(009) W408.07  ; 下料提升气缸下降
; rung 33
LD W400.03  ; 自动中
ANDNOT W390.00  ; 暂停 继续
AND W311.04  ; 下料提升气缸辅助1
AND W0.00  ; 手/自动切换HMI
AND 102.00  ; 放料停止拉带
RSET W311.04  ; 下料提升气缸辅助1
RSET 102.00  ; 放料停止拉带
RSET W412.00  ; 准备放右爪料
; rung 34: 放OK 下降 放料
STEP(008) W408.07  ; 下料提升气缸下降

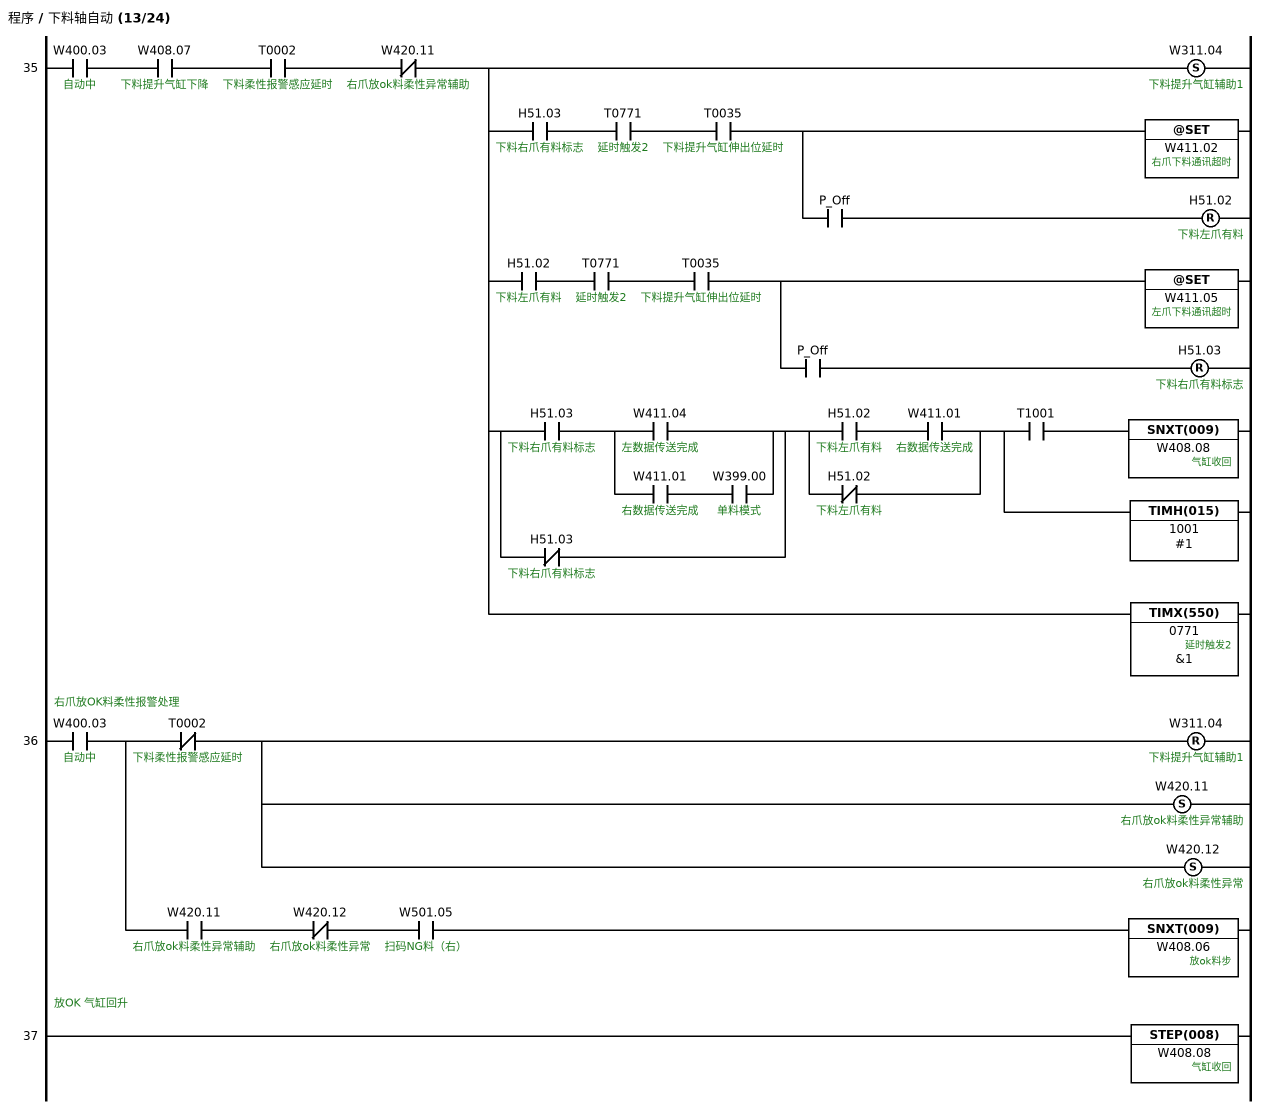
; rung 35
LD W400.03  ; 自动中
AND W408.07  ; 下料提升气缸下降
AND T0002  ; 下料柔性报警感应延时
ANDNOT W420.11  ; 右爪放ok料柔性异常辅助
OUT TR0
SET W311.04  ; 下料提升气缸辅助1
AND H51.03  ; 下料右爪有料标志
AND T0771  ; 延时触发2
AND T0035  ; 下料提升气缸伸出位延时
@SET W411.02  ; 右爪下料通讯超时
AND P_Off
RSET H51.02  ; 下料左爪有料
LD TR0
AND H51.02  ; 下料左爪有料
AND T0771  ; 延时触发2
AND T0035  ; 下料提升气缸伸出位延时
@SET W411.05  ; 左爪下料通讯超时
AND P_Off
RSET H51.03  ; 下料右爪有料标志
LD TR0
LD H51.03  ; 下料右爪有料标志
LD W411.04  ; 左数据传送完成
LD W411.01  ; 右数据传送完成
AND W399.00  ; 单料模式
ORLD
ANDLD
ORNOT H51.03  ; 下料右爪有料标志
ANDLD
LD H51.02  ; 下料左爪有料
AND W411.01  ; 右数据传送完成
ORNOT H51.02  ; 下料左爪有料
ANDLD
OUT TR1
AND T1001
SNXT(009) W408.08  ; 气缸收回
LD TR1
TIMH(015) 1001 #1
LD TR0
TIMX(550) 0771 &1  ; 延时触发2
; rung 36: 右爪放OK料柔性报警处理
LD W400.03  ; 自动中
OUT TR0
ANDNOT T0002  ; 下料柔性报警感应延时
RSET W311.04  ; 下料提升气缸辅助1
SET W420.11  ; 右爪放ok料柔性异常辅助
SET W420.12  ; 右爪放ok料柔性异常
LD TR0
AND W420.11  ; 右爪放ok料柔性异常辅助
ANDNOT W420.12  ; 右爪放ok料柔性异常
AND W501.05  ; 扫码NG料（右）
SNXT(009) W408.06  ; 放ok料步
; rung 37: 放OK 气缸回升
STEP(008) W408.08  ; 气缸收回

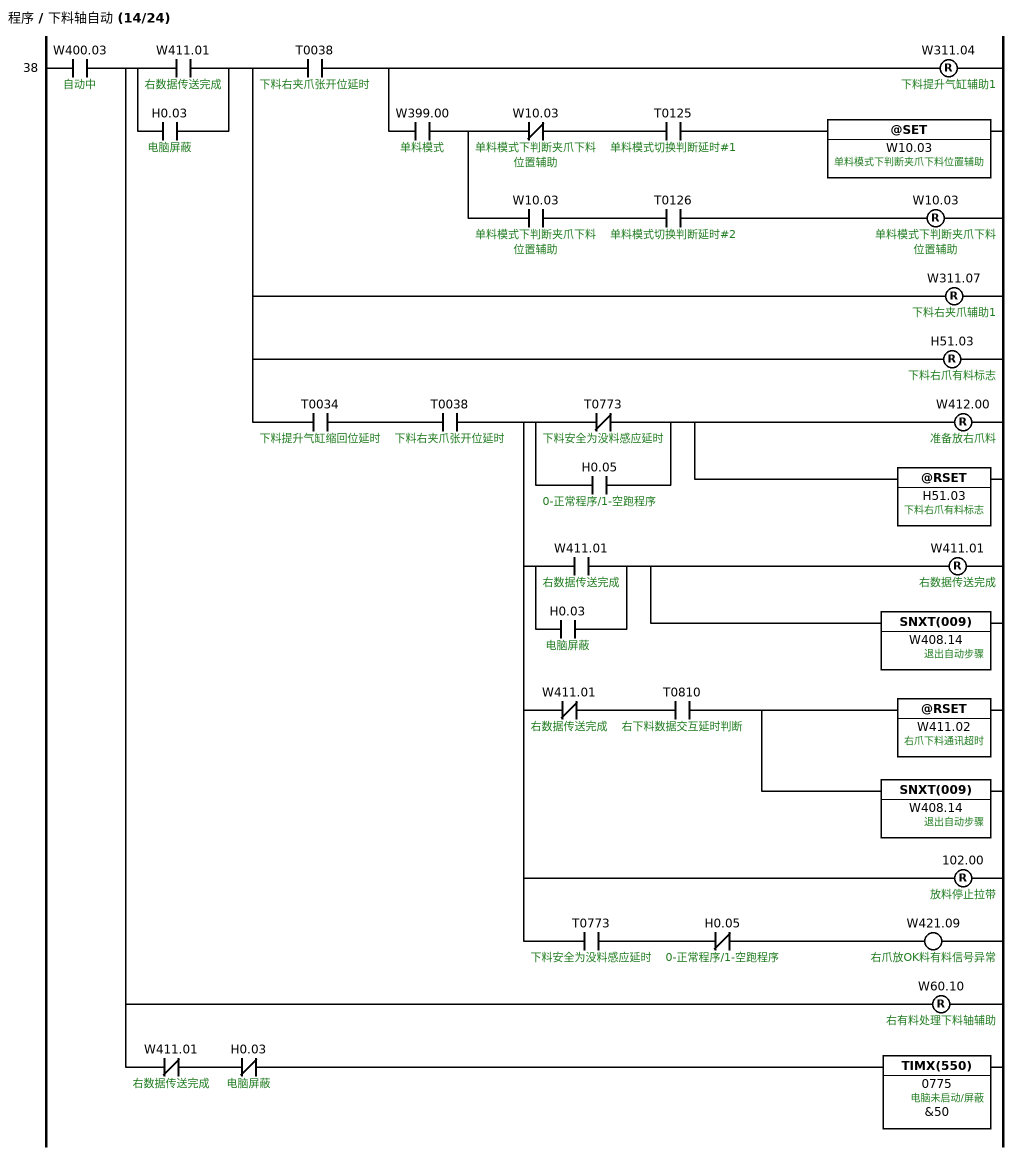
; rung 38
LD W400.03  ; 自动中
OUT TR0
LD W411.01  ; 右数据传送完成
OR H0.03  ; 电脑屏蔽
ANDLD
OUT TR1
AND T0038  ; 下料右夹爪张开位延时
RSET W311.04  ; 下料提升气缸辅助1
AND W399.00  ; 单料模式
OUT TR2
ANDNOT W10.03  ; 单料模式下判断夹爪下料位置辅助
AND T0125  ; 单料模式切换判断延时#1
@SET W10.03  ; 单料模式下判断夹爪下料位置辅助
LD TR2
AND W10.03  ; 单料模式下判断夹爪下料位置辅助
AND T0126  ; 单料模式切换判断延时#2
RSET W10.03  ; 单料模式下判断夹爪下料位置辅助
LD TR1
RSET W311.07  ; 下料右夹爪辅助1
RSET H51.03  ; 下料右爪有料标志
AND T0034  ; 下料提升气缸缩回位延时
AND T0038  ; 下料右夹爪张开位延时
OUT TR1
LDNOT T0773  ; 下料安全为没料感应延时
OR H0.05  ; 0-正常程序/1-空跑程序
ANDLD
RSET W412.00  ; 准备放右爪料
@RSET H51.03  ; 下料右爪有料标志
LD TR1
LD W411.01  ; 右数据传送完成
OR H0.03  ; 电脑屏蔽
ANDLD
RSET W411.01  ; 右数据传送完成
SNXT(009) W408.14  ; 退出自动步骤
LD TR1
ANDNOT W411.01  ; 右数据传送完成
AND T0810  ; 右下料数据交互延时判断
@RSET W411.02  ; 右爪下料通讯超时
SNXT(009) W408.14  ; 退出自动步骤
LD TR1
RSET 102.00  ; 放料停止拉带
AND T0773  ; 下料安全为没料感应延时
ANDNOT H0.05  ; 0-正常程序/1-空跑程序
OUT W421.09  ; 右爪放OK料有料信号异常
LD TR0
RSET W60.10  ; 右有料处理下料轴辅助
ANDNOT W411.01  ; 右数据传送完成
ANDNOT H0.03  ; 电脑屏蔽
TIMX(550) 0775 &50  ; 电脑未启动/屏蔽

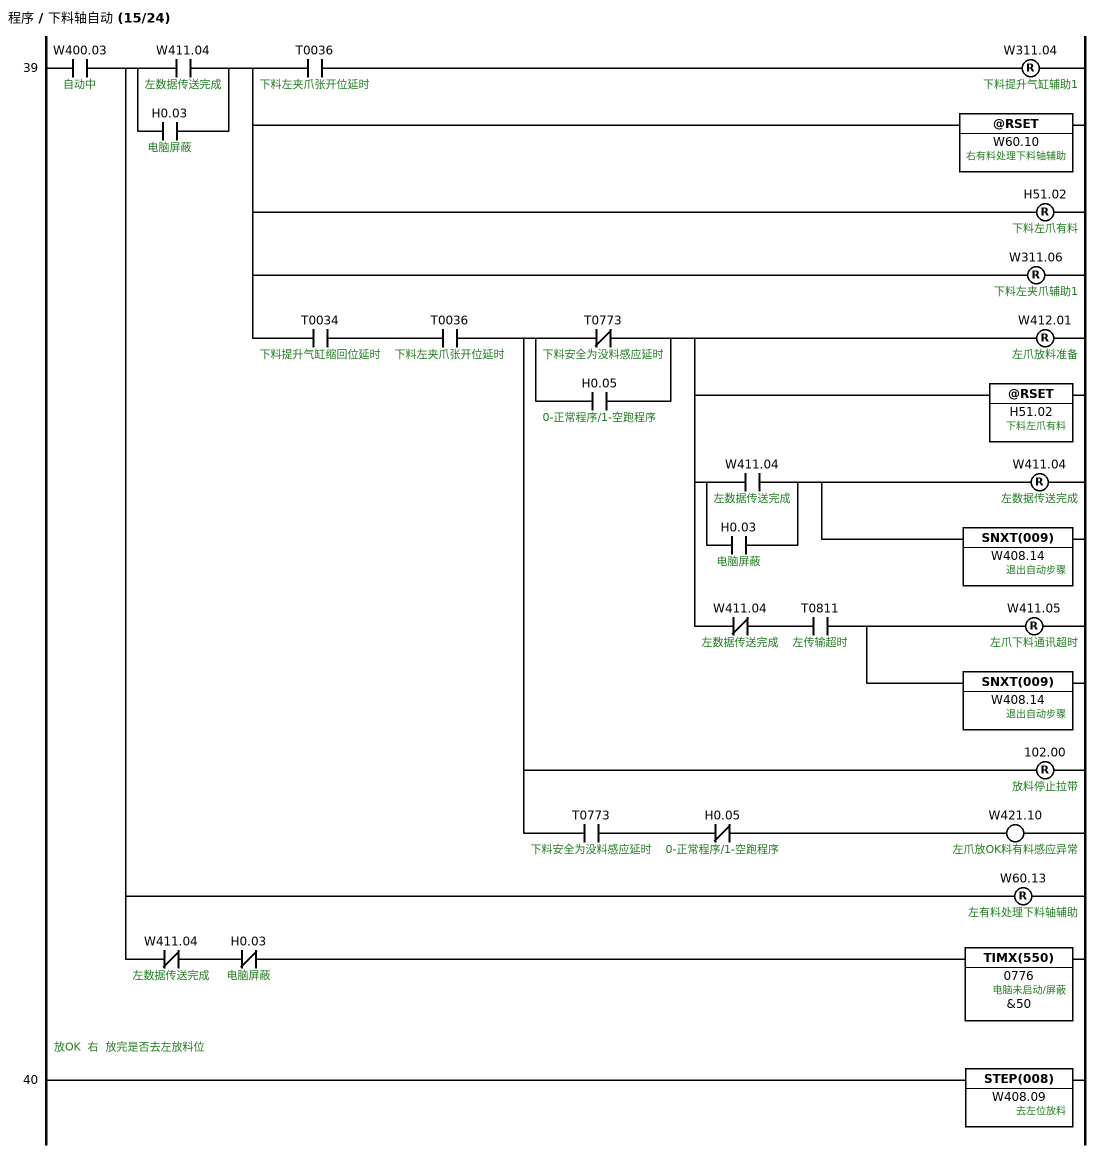
; rung 39
LD W400.03  ; 自动中
OUT TR0
LD W411.04  ; 左数据传送完成
OR H0.03  ; 电脑屏蔽
ANDLD
OUT TR1
AND T0036  ; 下料左夹爪张开位延时
RSET W311.04  ; 下料提升气缸辅助1
LD TR1
@RSET W60.10  ; 右有料处理下料轴辅助
RSET H51.02  ; 下料左爪有料
RSET W311.06  ; 下料左夹爪辅助1
AND T0034  ; 下料提升气缸缩回位延时
AND T0036  ; 下料左夹爪张开位延时
OUT TR1
LDNOT T0773  ; 下料安全为没料感应延时
OR H0.05  ; 0-正常程序/1-空跑程序
ANDLD
OUT TR2
RSET W412.01  ; 左爪放料准备
@RSET H51.02  ; 下料左爪有料
LD W411.04  ; 左数据传送完成
OR H0.03  ; 电脑屏蔽
ANDLD
RSET W411.04  ; 左数据传送完成
SNXT(009) W408.14  ; 退出自动步骤
LD TR2
ANDNOT W411.04  ; 左数据传送完成
AND T0811  ; 左传输超时
RSET W411.05  ; 左爪下料通讯超时
SNXT(009) W408.14  ; 退出自动步骤
LD TR1
RSET 102.00  ; 放料停止拉带
AND T0773  ; 下料安全为没料感应延时
ANDNOT H0.05  ; 0-正常程序/1-空跑程序
OUT W421.10  ; 左爪放OK料有料感应异常
LD TR0
RSET W60.13  ; 左有料处理下料轴辅助
ANDNOT W411.04  ; 左数据传送完成
ANDNOT H0.03  ; 电脑屏蔽
TIMX(550) 0776 &50  ; 电脑未启动/屏蔽
; rung 40: 放OK  右  放完是否去左放料位
STEP(008) W408.09  ; 去左位放料

